    S369_M_동작_선택_8 AT %MW5040.7 : BOOL; (* S369_M_동작_선택_8 *)
    S369_M_동작_선택_9 AT %MW5040.8 : BOOL; (* S369_M_동작_선택_9 *)
    S369_M_로딩_공정_불간섭 AT %MW5004.2 : BOOL; (* S369_M_공정_불간섭 *)
    S369_M_로딩_공정_원위치 AT %MW5004.0 : BOOL; (* S369_M_공정_원위치 *)
    S369_M_로딩_리셋보조 AT %MW5000.13 : BOOL;
    S369_M_로딩_이젝터_제품감지_무 AT %MW5001.9 : BOOL;
    S369_M_로딩_이젝터_제품감지_유 AT %MW5001.8 : BOOL;
    S369_M_로딩_작업_완료 AT %MW5001.0 : BOOL; (* S369_M_작업_완료 *)
    S369_M_로딩버퍼_SEQ AT %MW10240 : WORD; (* S369 M 로딩버퍼 SEQ *)
    S369_M_로딩버퍼_VIN_NO_1_2 AT %MW10251 : WORD; (* S369 M 로딩버퍼 VIN NO 1 2 *)
    S369_M_로딩버퍼_VIN_NO_3_4 AT %MW10252 : WORD; (* S369 M 로딩버퍼 VIN NO 3 4 *)
    S369_M_로딩버퍼_VIN_NO_5_6 AT %MW10253 : WORD; (* S369 M 로딩버퍼 VIN NO 5 6 *)
    S369_M_로딩버퍼_VIN_NO_7_8 AT %MW10254 : WORD; (* S369 M 로딩버퍼 VIN NO 7 8 *)
    S369_M_로딩버퍼_VIN_NO_9_10 AT %MW10255 : WORD; (* S369 M 로딩버퍼 VIN NO 9 10 *)
    S369_M_로딩버퍼_제품감지_무 AT %MW5005.1 : BOOL; (* S369_로딩버퍼_제품감지_무 *)
    S369_M_로딩버퍼_제품감지_유 AT %MW5005.0 : BOOL; (* S369_로딩버퍼_제품감지_유 *)
    S369_M_로딩버퍼_차종1_AX AT %MW10241.0 : BOOL; (* S369 M 로딩버퍼 차종1 AX *)
    S369_M_로딩버퍼_차종1_B AT %MW10241.1 : BOOL; (* S369 M 로딩버퍼 차종1 B *)
    S369_M_로딩버퍼_차종1_C AT %MW10241.2 : BOOL; (* S369 M 로딩버퍼 차종1 C *)
    S369_M_로딩버퍼_차종1_D AT %MW10241.3 : BOOL; (* S369 M 로딩버퍼 차종1 D *)
    S369_M_로딩버퍼_차종1_E AT %MW10241.4 : BOOL; (* S369 M 로딩버퍼 차종1 E *)
    S369_M_로딩버퍼_차종1_F AT %MW10241.5 : BOOL; (* S369 M 로딩버퍼 차종1 F *)
    S369_M_로딩버퍼_차종1_G AT %MW10241.6 : BOOL; (* S369 M 로딩버퍼 차종1 G *)
    S369_M_로딩버퍼_차종1_H AT %MW10241.7 : BOOL; (* S369 M 로딩버퍼 차종1 H *)
    S369_M_로딩버퍼_차종2_3DR AT %MW10241.8 : BOOL; (* S369 M 로딩버퍼 차종2 3DR *)
    S369_M_로딩버퍼_차종2_4DR AT %MW10241.9 : BOOL; (* S369 M 로딩버퍼 차종2 4DR *)
    S369_M_로딩버퍼_차종2_5DR AT %MW10241.10 : BOOL; (* S369 M 로딩버퍼 차종2 5DR *)
    S369_M_로딩버퍼_차종2_SP1 AT %MW10241.12 : BOOL; (* S369 M 로딩버퍼 차종2 SP1 *)
    S369_M_로딩버퍼_차종2_SP2 AT %MW10241.13 : BOOL; (* S369 M 로딩버퍼 차종2 SP2 *)
    S369_M_로딩버퍼_차종2_WGN AT %MW10241.11 : BOOL; (* S369 M 로딩버퍼 차종2 WGN *)
    S369_M_로딩버퍼_차종3_LHD AT %MW10241.14 : BOOL; (* S369 M 로딩버퍼 차종3 LHD *)
    S369_M_로딩버퍼_차종3_RHD AT %MW10241.15 : BOOL; (* S369 M 로딩버퍼 차종3 RHD *)
    S369_M_로딩버퍼_차종4_EEC AT %MW10242.3 : BOOL; (* S369 M 로딩버퍼 차종4 EEC *)
    S369_M_로딩버퍼_차종4_SP1 AT %MW10242.8 : BOOL; (* S369 M 로딩버퍼 차종4 SP1 *)
    S369_M_로딩버퍼_차종4_SP2 AT %MW10242.9 : BOOL; (* S369 M 로딩버퍼 차종4 SP2 *)
    S369_M_로딩버퍼_차종4_SP3 AT %MW10242.11 : BOOL; (* S369 M 로딩버퍼 차종4 SP3 *)
    S369_M_로딩버퍼_차종4_SP4 AT %MW10242.12 : BOOL; (* S369 M 로딩버퍼 차종4 SP4 *)
    S369_M_로딩버퍼_차종4_SP5 AT %MW10242.13 : BOOL; (* S369 M 로딩버퍼 차종4 SP5 *)
    S369_M_로딩버퍼_차종4_SP6 AT %MW10242.14 : BOOL; (* S369 M 로딩버퍼 차종4 SP6 *)
    S369_M_로딩버퍼_차종4_SP7 AT %MW10242.15 : BOOL; (* S369 M 로딩버퍼 차종4 SP7 *)
    S369_M_로딩버퍼_차종4_내수 AT %MW10242.0 : BOOL; (* S369 M 로딩버퍼 차종4 내수 *)
    S369_M_로딩버퍼_차종4_러시아 AT %MW10242.10 : BOOL; (* S369 M 로딩버퍼 차종4 러시아 *)
    S369_M_로딩버퍼_차종4_북미 AT %MW10242.2 : BOOL; (* S369 M 로딩버퍼 차종4 북미 *)
    S369_M_로딩버퍼_차종4_브라질 AT %MW10242.7 : BOOL; (* S369 M 로딩버퍼 차종4 브라질 *)
    S369_M_로딩버퍼_차종4_수출 AT %MW10242.1 : BOOL; (* S369 M 로딩버퍼 차종4 수출 *)
    S369_M_로딩버퍼_차종4_중국 AT %MW10242.6 : BOOL; (* S369 M 로딩버퍼 차종4 중국 *)
    S369_M_로딩버퍼_차종4_중동 AT %MW10242.5 : BOOL; (* S369 M 로딩버퍼 차종4 중동 *)
    S369_M_로딩버퍼_차종4_호주 AT %MW10242.4 : BOOL; (* S369 M 로딩버퍼 차종4 호주 *)
    S369_M_로딩버퍼_차종5_AT AT %MW10243.1 : BOOL; (* S369 M 로딩버퍼 차종5 AT *)
    S369_M_로딩버퍼_차종5_MT AT %MW10243.0 : BOOL; (* S369 M 로딩버퍼 차종5 MT *)
    S369_M_로딩버퍼_차종5_SP1 AT %MW10243.2 : BOOL; (* S369 M 로딩버퍼 차종5 SP1 *)
    S369_M_로딩버퍼_차종6_DSROOF AT %MW10243.6 : BOOL; (* S369 M 로딩버퍼 차종6 DSROOF *)
    S369_M_로딩버퍼_차종6_SP1 AT %MW10243.7 : BOOL; (* S369 M 로딩버퍼 차종6 SP1 *)
    S369_M_로딩버퍼_차종6_썬루프 AT %MW10243.4 : BOOL; (* S369 M 로딩버퍼 차종6 썬루프 *)
    S369_M_로딩버퍼_차종6_일반루프 AT %MW10243.3 : BOOL; (* S369 M 로딩버퍼 차종6 일반루프 *)
    S369_M_로딩버퍼_차종6_파노라마루프 AT %MW10243.5 : BOOL; (* S369 M 로딩버퍼 차종6 파노라마루프 *)
    S369_M_로딩버퍼_차종7_DSL AT %MW10243.9 : BOOL; (* S369 M 로딩버퍼 차종7 DSL *)
    S369_M_로딩버퍼_차종7_GSL AT %MW10243.8 : BOOL; (* S369 M 로딩버퍼 차종7 GSL *)
    S369_M_로딩버퍼_차종7_SP1 AT %MW10243.10 : BOOL; (* S369 M 로딩버퍼 차종7 SP1 *)
    S369_M_로딩버퍼_차종7_SP2 AT %MW10243.11 : BOOL; (* S369 M 로딩버퍼 차종7 SP2 *)
    S369_M_로딩버퍼_차종7_SP3 AT %MW10243.12 : BOOL; (* S369 M 로딩버퍼 차종7 SP3 *)
    S369_M_로딩버퍼_차종7_SP4 AT %MW10243.13 : BOOL; (* S369 M 로딩버퍼 차종7 SP4 *)
    S369_M_로딩버퍼_차종7_SP5 AT %MW10243.14 : BOOL; (* S369 M 로딩버퍼 차종7 SP5 *)
    S369_M_로딩버퍼_차종7_SP6 AT %MW10243.15 : BOOL; (* S369 M 로딩버퍼 차종7 SP6 *)
    S369_M_로딩버퍼_차종8_2WD AT %MW10244.0 : BOOL; (* S369 M 로딩버퍼 차종8 2WD *)
    S369_M_로딩버퍼_차종8_4WD AT %MW10244.1 : BOOL; (* S369 M 로딩버퍼 차종8 4WD *)
    S369_M_로딩버퍼_차종8_SP1 AT %MW10244.2 : BOOL; (* S369 M 로딩버퍼 차종8 SP1 *)
    S369_M_로딩버퍼_차종9_MPI AT %MW10244.3 : BOOL; (* S369 M 로딩버퍼 차종9 MPI *)
    S369_M_로딩버퍼_차종9_SP1 AT %MW10244.5 : BOOL; (* S369 M 로딩버퍼 차종9 SP1 *)
    S369_M_로딩버퍼_차종9_SP10 AT %MW10244.14 : BOOL; (* S369 M 로딩버퍼 차종9 SP10 *)
    S369_M_로딩버퍼_차종9_SP11 AT %MW10244.15 : BOOL; (* S369 M 로딩버퍼 차종9 SP11 *)
    S369_M_로딩버퍼_차종9_SP2 AT %MW10244.6 : BOOL; (* S369 M 로딩버퍼 차종9 SP2 *)
    S369_M_로딩버퍼_차종9_SP3 AT %MW10244.7 : BOOL; (* S369 M 로딩버퍼 차종9 SP3 *)
    S369_M_로딩버퍼_차종9_SP4 AT %MW10244.8 : BOOL; (* S369 M 로딩버퍼 차종9 SP4 *)
    S369_M_로딩버퍼_차종9_SP5 AT %MW10244.9 : BOOL; (* S369 M 로딩버퍼 차종9 SP5 *)
    S369_M_로딩버퍼_차종9_SP6 AT %MW10244.10 : BOOL; (* S369 M 로딩버퍼 차종9 SP6 *)
    S369_M_로딩버퍼_차종9_SP7 AT %MW10244.11 : BOOL; (* S369 M 로딩버퍼 차종9 SP7 *)
    S369_M_로딩버퍼_차종9_SP8 AT %MW10244.12 : BOOL; (* S369 M 로딩버퍼 차종9 SP8 *)
    S369_M_로딩버퍼_차종9_SP9 AT %MW10244.13 : BOOL; (* S369 M 로딩버퍼 차종9 SP9 *)
    S369_M_로딩버퍼_차종9_T_GDI AT %MW10244.4 : BOOL; (* S369 M 로딩버퍼 차종9 T GDI *)
    S369_M_로딩버퍼_차종_AS AT %MW10250.9 : BOOL; (* S369 M 로딩버퍼 차종 AS *)
    S369_M_로딩버퍼_차종_OPT1_R_RACK_무 AT %MW10245.3 : BOOL; (* S369 M 로딩버퍼 차종 OPT1 R RACK 무 *)
    S369_M_로딩버퍼_차종_OPT1_R_RACK_유 AT %MW10245.2 : BOOL; (* S369 M 로딩버퍼 차종 OPT1 R RACK 유 *)
    S369_M_로딩버퍼_차종_OPT1_SP1 AT %MW10245.10 : BOOL; (* S369 M 로딩버퍼 차종 OPT1 SP1 *)
    S369_M_로딩버퍼_차종_OPT1_SP2 AT %MW10245.11 : BOOL; (* S369 M 로딩버퍼 차종 OPT1 SP2 *)
    S369_M_로딩버퍼_차종_OPT1_SP3 AT %MW10245.12 : BOOL; (* S369 M 로딩버퍼 차종 OPT1 SP3 *)
    S369_M_로딩버퍼_차종_OPT1_SP4 AT %MW10245.13 : BOOL; (* S369 M 로딩버퍼 차종 OPT1 SP4 *)
    S369_M_로딩버퍼_차종_OPT1_SP5 AT %MW10245.14 : BOOL; (* S369 M 로딩버퍼 차종 OPT1 SP5 *)
    S369_M_로딩버퍼_차종_OPT1_SP6 AT %MW10245.15 : BOOL; (* S369 M 로딩버퍼 차종 OPT1 SP6 *)
    S369_M_로딩버퍼_차종_OPT1_S_REP_EATER_무 AT %MW10245.7 : BOOL; (* S369 M 로딩버퍼 차종 OPT1 S REP EATER 무 *)
    S369_M_로딩버퍼_차종_OPT1_S_REP_EATER_유 AT %MW10245.6 : BOOL; (* S369 M 로딩버퍼 차종 OPT1 S REP EATER 유 *)
    S369_M_로딩버퍼_차종_OPT1_VAN_무 AT %MW10245.9 : BOOL; (* S369 M 로딩버퍼 차종 OPT1 VAN 무 *)
    S369_M_로딩버퍼_차종_OPT1_VAN_유 AT %MW10245.8 : BOOL; (* S369 M 로딩버퍼 차종 OPT1 VAN 유 *)
    S369_M_로딩버퍼_차종_OPT1_슬라이딩_무 AT %MW10245.1 : BOOL; (* S369 M 로딩버퍼 차종 OPT1 슬라이딩 무 *)
    S369_M_로딩버퍼_차종_OPT1_슬라이딩_유 AT %MW10245.0 : BOOL; (* S369 M 로딩버퍼 차종 OPT1 슬라이딩 유 *)
    S369_M_로딩버퍼_차종_OPT1_폴딩_무 AT %MW10245.5 : BOOL; (* S369 M 로딩버퍼 차종 OPT1 폴딩 무 *)
    S369_M_로딩버퍼_차종_OPT1_폴딩_유 AT %MW10245.4 : BOOL; (* S369 M 로딩버퍼 차종 OPT1 폴딩 유 *)
    S369_M_로딩버퍼_차종_OPT2_SP_WORD1 AT %MW10246 : WORD; (* S369 M 로딩버퍼 차종 OPT2 SP WORD1 *)
    S369_M_로딩버퍼_차종_OPT3_SP_WORD2 AT %MW10247 : WORD; (* S369 M 로딩버퍼 차종 OPT3 SP WORD2 *)
    S369_M_로딩버퍼_차종_OPT4_SP_WORD3 AT %MW10248 : WORD; (* S369 M 로딩버퍼 차종 OPT4 SP WORD3 *)
    S369_M_로딩버퍼_차종_OPT5_SP_WORD4 AT %MW10249 : WORD; (* S369 M 로딩버퍼 차종 OPT5 SP WORD4 *)
    S369_M_로딩버퍼_차종_SP1 AT %MW10250.0 : BOOL; (* S369 M 로딩버퍼 차종 SP1 *)
    S369_M_로딩버퍼_차종_SP2 AT %MW10250.1 : BOOL; (* S369 M 로딩버퍼 차종 SP2 *)
    S369_M_로딩버퍼_차종_SP3 AT %MW10250.2 : BOOL; (* S369 M 로딩버퍼 차종 SP3 *)
    S369_M_로딩버퍼_차종_SP4 AT %MW10250.3 : BOOL; (* S369 M 로딩버퍼 차종 SP4 *)
    S369_M_로딩버퍼_차종_SP5 AT %MW10250.4 : BOOL; (* S369 M 로딩버퍼 차종 SP5 *)
    S369_M_로딩버퍼_차종_SP6 AT %MW10250.5 : BOOL; (* S369 M 로딩버퍼 차종 SP6 *)
    S369_M_로딩버퍼_차종_SP7 AT %MW10250.6 : BOOL; (* S369 M 로딩버퍼 차종 SP7 *)
    S369_M_로딩버퍼_차종_SP8 AT %MW10250.7 : BOOL; (* S369 M 로딩버퍼 차종 SP8 *)
    S369_M_로딩버퍼_차종_SP9 AT %MW10250.15 : BOOL; (* S369 M 로딩버퍼 차종 SP9 *)
    S369_M_로딩버퍼_차종_공대차 AT %MW10250.12 : BOOL; (* S369 M 로딩버퍼 차종 공대차 *)
    S369_M_로딩버퍼_차종_공차 AT %MW10250.10 : BOOL; (* S369 M 로딩버퍼 차종 공차 *)
    S369_M_로딩버퍼_차종_무 AT %MW5002.1 : BOOL;
    S369_M_로딩버퍼_차종_불량대차 AT %MW10250.13 : BOOL; (* S369 M 로딩버퍼 차종 불량대차 *)
    S369_M_로딩버퍼_차종_불량차 AT %MW10250.11 : BOOL; (* S369 M 로딩버퍼 차종 불량차 *)
    S369_M_로딩버퍼_차종_비축 AT %MW10250.8 : BOOL; (* S369 M 로딩버퍼 차종 비축 *)
    S369_M_로딩버퍼_차종_유 AT %MW5002.0 : BOOL;
    S369_M_로딩버퍼_차종_취출대차 AT %MW10250.14 : BOOL; (* S369 M 로딩버퍼 차종 취출대차 *)
    S369_M_부저_정지_보조 AT %MW5000.11 : BOOL; (* S369_M_부저_정지_보조 *)
    S369_M_수동모드 AT %MW5000.3 : BOOL; (* S369 선택 수동모드 *)
    S369_M_언로딩_공정_불간섭 AT %MW5004.3 : BOOL;
    S369_M_언로딩_공정_원위치 AT %MW5004.1 : BOOL;
    S369_M_언로딩_이젝터_제품감지_무 AT %MW5001.11 : BOOL;
    S369_M_언로딩_이젝터_제품감지_유 AT %MW5001.10 : BOOL;
    S369_M_언로딩_작업_완료 AT %MW5001.1 : BOOL;
    S369_M_언로딩버퍼_SEQ AT %MW10340 : WORD; (* S369 M 언로딩버퍼 SEQ *)
    S369_M_언로딩버퍼_VIN_NO_1_2 AT %MW10351 : WORD; (* S369 M 언로딩버퍼 VIN NO 1 2 *)
    S369_M_언로딩버퍼_VIN_NO_3_4 AT %MW10352 : WORD; (* S369 M 언로딩버퍼 VIN NO 3 4 *)
    S369_M_언로딩버퍼_VIN_NO_5_6 AT %MW10353 : WORD; (* S369 M 언로딩버퍼 VIN NO 5 6 *)
    S369_M_언로딩버퍼_VIN_NO_7_8 AT %MW10354 : WORD; (* S369 M 언로딩버퍼 VIN NO 7 8 *)
    S369_M_언로딩버퍼_VIN_NO_9_10 AT %MW10355 : WORD; (* S369 M 언로딩버퍼 VIN NO 9 10 *)
    S369_M_언로딩버퍼_도착완료 AT %MW5003.6 : BOOL;
    S369_M_언로딩버퍼_제품감지_무 AT %MW5005.11 : BOOL; (* S369_언로딩버퍼_제품감지_무 *)
    S369_M_언로딩버퍼_제품감지_유 AT %MW5005.10 : BOOL; (* S369_언로딩버퍼_제품감지_유 *)
    S369_M_언로딩버퍼_차종1_AX AT %MW10341.0 : BOOL; (* S369 M 언로딩버퍼 차종1 AX *)
    S369_M_언로딩버퍼_차종1_B AT %MW10341.1 : BOOL; (* S369 M 언로딩버퍼 차종1 B *)
    S369_M_언로딩버퍼_차종1_C AT %MW10341.2 : BOOL; (* S369 M 언로딩버퍼 차종1 C *)
    S369_M_언로딩버퍼_차종1_D AT %MW10341.3 : BOOL; (* S369 M 언로딩버퍼 차종1 D *)
    S369_M_언로딩버퍼_차종1_E AT %MW10341.4 : BOOL; (* S369 M 언로딩버퍼 차종1 E *)
    S369_M_언로딩버퍼_차종1_F AT %MW10341.5 : BOOL; (* S369 M 언로딩버퍼 차종1 F *)
    S369_M_언로딩버퍼_차종1_G AT %MW10341.6 : BOOL; (* S369 M 언로딩버퍼 차종1 G *)
    S369_M_언로딩버퍼_차종1_H AT %MW10341.7 : BOOL; (* S369 M 언로딩버퍼 차종1 H *)
    S369_M_언로딩버퍼_차종2_3DR AT %MW10341.8 : BOOL; (* S369 M 언로딩버퍼 차종2 3DR *)
    S369_M_언로딩버퍼_차종2_4DR AT %MW10341.9 : BOOL; (* S369 M 언로딩버퍼 차종2 4DR *)
    S369_M_언로딩버퍼_차종2_5DR AT %MW10341.10 : BOOL; (* S369 M 언로딩버퍼 차종2 5DR *)
    S369_M_언로딩버퍼_차종2_SP1 AT %MW10341.12 : BOOL; (* S369 M 언로딩버퍼 차종2 SP1 *)
    S369_M_언로딩버퍼_차종2_SP2 AT %MW10341.13 : BOOL; (* S369 M 언로딩버퍼 차종2 SP2 *)
    S369_M_언로딩버퍼_차종2_WGN AT %MW10341.11 : BOOL; (* S369 M 언로딩버퍼 차종2 WGN *)
    S369_M_언로딩버퍼_차종3_LHD AT %MW10341.14 : BOOL; (* S369 M 언로딩버퍼 차종3 LHD *)
    S369_M_언로딩버퍼_차종3_RHD AT %MW10341.15 : BOOL; (* S369 M 언로딩버퍼 차종3 RHD *)
    S369_M_언로딩버퍼_차종4_EEC AT %MW10342.3 : BOOL; (* S369 M 언로딩버퍼 차종4 EEC *)
    S369_M_언로딩버퍼_차종4_SP1 AT %MW10342.8 : BOOL; (* S369 M 언로딩버퍼 차종4 SP1 *)
    S369_M_언로딩버퍼_차종4_SP2 AT %MW10342.9 : BOOL; (* S369 M 언로딩버퍼 차종4 SP2 *)
    S369_M_언로딩버퍼_차종4_SP3 AT %MW10342.11 : BOOL; (* S369 M 언로딩버퍼 차종4 SP3 *)
    S369_M_언로딩버퍼_차종4_SP4 AT %MW10342.12 : BOOL; (* S369 M 언로딩버퍼 차종4 SP4 *)
    S369_M_언로딩버퍼_차종4_SP5 AT %MW10342.13 : BOOL; (* S369 M 언로딩버퍼 차종4 SP5 *)
    S369_M_언로딩버퍼_차종4_SP6 AT %MW10342.14 : BOOL; (* S369 M 언로딩버퍼 차종4 SP6 *)
    S369_M_언로딩버퍼_차종4_SP7 AT %MW10342.15 : BOOL; (* S369 M 언로딩버퍼 차종4 SP7 *)
    S369_M_언로딩버퍼_차종4_내수 AT %MW10342.0 : BOOL; (* S369 M 언로딩버퍼 차종4 내수 *)
    S369_M_언로딩버퍼_차종4_러시아 AT %MW10342.10 : BOOL; (* S369 M 언로딩버퍼 차종4 러시아 *)
    S369_M_언로딩버퍼_차종4_북미 AT %MW10342.2 : BOOL; (* S369 M 언로딩버퍼 차종4 북미 *)
    S369_M_언로딩버퍼_차종4_브라질 AT %MW10342.7 : BOOL; (* S369 M 언로딩버퍼 차종4 브라질 *)
    S369_M_언로딩버퍼_차종4_수출 AT %MW10342.1 : BOOL; (* S369 M 언로딩버퍼 차종4 수출 *)
    S369_M_언로딩버퍼_차종4_중국 AT %MW10342.6 : BOOL; (* S369 M 언로딩버퍼 차종4 중국 *)
    S369_M_언로딩버퍼_차종4_중동 AT %MW10342.5 : BOOL; (* S369 M 언로딩버퍼 차종4 중동 *)
    S369_M_언로딩버퍼_차종4_호주 AT %MW10342.4 : BOOL; (* S369 M 언로딩버퍼 차종4 호주 *)
    S369_M_언로딩버퍼_차종5_AT AT %MW10343.1 : BOOL; (* S369 M 언로딩버퍼 차종5 AT *)
    S369_M_언로딩버퍼_차종5_MT AT %MW10343.0 : BOOL; (* S369 M 언로딩버퍼 차종5 MT *)
    S369_M_언로딩버퍼_차종5_SP1 AT %MW10343.2 : BOOL; (* S369 M 언로딩버퍼 차종5 SP1 *)
    S369_M_언로딩버퍼_차종6_DSROOF AT %MW10343.6 : BOOL; (* S369 M 언로딩버퍼 차종6 DSROOF *)
    S369_M_언로딩버퍼_차종6_SP1 AT %MW10343.7 : BOOL; (* S369 M 언로딩버퍼 차종6 SP1 *)
    S369_M_언로딩버퍼_차종6_썬루프 AT %MW10343.4 : BOOL; (* S369 M 언로딩버퍼 차종6 썬루프 *)
    S369_M_언로딩버퍼_차종6_일반루프 AT %MW10343.3 : BOOL; (* S369 M 언로딩버퍼 차종6 일반루프 *)
    S369_M_언로딩버퍼_차종6_파노라마루프 AT %MW10343.5 : BOOL; (* S369 M 언로딩버퍼 차종6 파노라마루프 *)
    S369_M_언로딩버퍼_차종7_DSL AT %MW10343.9 : BOOL; (* S369 M 언로딩버퍼 차종7 DSL *)
    S369_M_언로딩버퍼_차종7_GSL AT %MW10343.8 : BOOL; (* S369 M 언로딩버퍼 차종7 GSL *)
    S369_M_언로딩버퍼_차종7_SP1 AT %MW10343.10 : BOOL; (* S369 M 언로딩버퍼 차종7 SP1 *)
    S369_M_언로딩버퍼_차종7_SP2 AT %MW10343.11 : BOOL; (* S369 M 언로딩버퍼 차종7 SP2 *)
    S369_M_언로딩버퍼_차종7_SP3 AT %MW10343.12 : BOOL; (* S369 M 언로딩버퍼 차종7 SP3 *)
    S369_M_언로딩버퍼_차종7_SP4 AT %MW10343.13 : BOOL; (* S369 M 언로딩버퍼 차종7 SP4 *)
    S369_M_언로딩버퍼_차종7_SP5 AT %MW10343.14 : BOOL; (* S369 M 언로딩버퍼 차종7 SP5 *)
    S369_M_언로딩버퍼_차종7_SP6 AT %MW10343.15 : BOOL; (* S369 M 언로딩버퍼 차종7 SP6 *)
    S369_M_언로딩버퍼_차종8_2WD AT %MW10344.0 : BOOL; (* S369 M 언로딩버퍼 차종8 2WD *)
    S369_M_언로딩버퍼_차종8_4WD AT %MW10344.1 : BOOL; (* S369 M 언로딩버퍼 차종8 4WD *)
    S369_M_언로딩버퍼_차종8_SP1 AT %MW10344.2 : BOOL; (* S369 M 언로딩버퍼 차종8 SP1 *)
    S369_M_언로딩버퍼_차종9_MPI AT %MW10344.3 : BOOL; (* S369 M 언로딩버퍼 차종9 MPI *)
    S369_M_언로딩버퍼_차종9_SP1 AT %MW10344.5 : BOOL; (* S369 M 언로딩버퍼 차종9 SP1 *)
    S369_M_언로딩버퍼_차종9_SP10 AT %MW10344.14 : BOOL; (* S369 M 언로딩버퍼 차종9 SP10 *)
    S369_M_언로딩버퍼_차종9_SP11 AT %MW10344.15 : BOOL; (* S369 M 언로딩버퍼 차종9 SP11 *)
    S369_M_언로딩버퍼_차종9_SP2 AT %MW10344.6 : BOOL; (* S369 M 언로딩버퍼 차종9 SP2 *)
    S369_M_언로딩버퍼_차종9_SP3 AT %MW10344.7 : BOOL; (* S369 M 언로딩버퍼 차종9 SP3 *)
    S369_M_언로딩버퍼_차종9_SP4 AT %MW10344.8 : BOOL; (* S369 M 언로딩버퍼 차종9 SP4 *)
    S369_M_언로딩버퍼_차종9_SP5 AT %MW10344.9 : BOOL; (* S369 M 언로딩버퍼 차종9 SP5 *)
    S369_M_언로딩버퍼_차종9_SP6 AT %MW10344.10 : BOOL; (* S369 M 언로딩버퍼 차종9 SP6 *)
    S369_M_언로딩버퍼_차종9_SP7 AT %MW10344.11 : BOOL; (* S369 M 언로딩버퍼 차종9 SP7 *)
    S369_M_언로딩버퍼_차종9_SP8 AT %MW10344.12 : BOOL; (* S369 M 언로딩버퍼 차종9 SP8 *)
    S369_M_언로딩버퍼_차종9_SP9 AT %MW10344.13 : BOOL; (* S369 M 언로딩버퍼 차종9 SP9 *)
    S369_M_언로딩버퍼_차종9_T_GDI AT %MW10344.4 : BOOL; (* S369 M 언로딩버퍼 차종9 T GDI *)
    S369_M_언로딩버퍼_차종_AS AT %MW10350.9 : BOOL; (* S369 M 언로딩버퍼 차종 AS *)
    S369_M_언로딩버퍼_차종_OPT1_R_RACK_무 AT %MW10345.3 : BOOL; (* S369 M 언로딩버퍼 차종 OPT1 R RACK 무 *)
    S369_M_언로딩버퍼_차종_OPT1_R_RACK_유 AT %MW10345.2 : BOOL; (* S369 M 언로딩버퍼 차종 OPT1 R RACK 유 *)
    S369_M_언로딩버퍼_차종_OPT1_SP1 AT %MW10345.10 : BOOL; (* S369 M 언로딩버퍼 차종 OPT1 SP1 *)
    S369_M_언로딩버퍼_차종_OPT1_SP2 AT %MW10345.11 : BOOL; (* S369 M 언로딩버퍼 차종 OPT1 SP2 *)
    S369_M_언로딩버퍼_차종_OPT1_SP3 AT %MW10345.12 : BOOL; (* S369 M 언로딩버퍼 차종 OPT1 SP3 *)
    S369_M_언로딩버퍼_차종_OPT1_SP4 AT %MW10345.13 : BOOL; (* S369 M 언로딩버퍼 차종 OPT1 SP4 *)
    S369_M_언로딩버퍼_차종_OPT1_SP5 AT %MW10345.14 : BOOL; (* S369 M 언로딩버퍼 차종 OPT1 SP5 *)
    S369_M_언로딩버퍼_차종_OPT1_SP6 AT %MW10345.15 : BOOL; (* S369 M 언로딩버퍼 차종 OPT1 SP6 *)
    S369_M_언로딩버퍼_차종_OPT1_S_REP_EATER_무 AT %MW10345.7 : BOOL; (* S369 M 언로딩버퍼 차종 OPT1 S REP EATER 무 *)
    S369_M_언로딩버퍼_차종_OPT1_S_REP_EATER_유 AT %MW10345.6 : BOOL; (* S369 M 언로딩버퍼 차종 OPT1 S REP EATER 유 *)
    S369_M_언로딩버퍼_차종_OPT1_VAN_무 AT %MW10345.9 : BOOL; (* S369 M 언로딩버퍼 차종 OPT1 VAN 무 *)
    S369_M_언로딩버퍼_차종_OPT1_VAN_유 AT %MW10345.8 : BOOL; (* S369 M 언로딩버퍼 차종 OPT1 VAN 유 *)
    S369_M_언로딩버퍼_차종_OPT1_슬라이딩_무 AT %MW10345.1 : BOOL; (* S369 M 언로딩버퍼 차종 OPT1 슬라이딩 무 *)
    S369_M_언로딩버퍼_차종_OPT1_슬라이딩_유 AT %MW10345.0 : BOOL; (* S369 M 언로딩버퍼 차종 OPT1 슬라이딩 유 *)
    S369_M_언로딩버퍼_차종_OPT1_폴딩_무 AT %MW10345.5 : BOOL; (* S369 M 언로딩버퍼 차종 OPT1 폴딩 무 *)
    S369_M_언로딩버퍼_차종_OPT1_폴딩_유 AT %MW10345.4 : BOOL; (* S369 M 언로딩버퍼 차종 OPT1 폴딩 유 *)
    S369_M_언로딩버퍼_차종_OPT2_SP_WORD1 AT %MW10346 : WORD; (* S369 M 언로딩버퍼 차종 OPT2 SP WORD1 *)
    S369_M_언로딩버퍼_차종_OPT3_SP_WORD2 AT %MW10347 : WORD; (* S369 M 언로딩버퍼 차종 OPT3 SP WORD2 *)
    S369_M_언로딩버퍼_차종_OPT4_SP_WORD3 AT %MW10348 : WORD; (* S369 M 언로딩버퍼 차종 OPT4 SP WORD3 *)
    S369_M_언로딩버퍼_차종_OPT5_SP_WORD4 AT %MW10349 : WORD; (* S369 M 언로딩버퍼 차종 OPT5 SP WORD4 *)
    S369_M_언로딩버퍼_차종_SP1 AT %MW10350.0 : BOOL; (* S369 M 언로딩버퍼 차종 SP1 *)
    S369_M_언로딩버퍼_차종_SP2 AT %MW10350.1 : BOOL; (* S369 M 언로딩버퍼 차종 SP2 *)
    S369_M_언로딩버퍼_차종_SP3 AT %MW10350.2 : BOOL; (* S369 M 언로딩버퍼 차종 SP3 *)
    S369_M_언로딩버퍼_차종_SP4 AT %MW10350.3 : BOOL; (* S369 M 언로딩버퍼 차종 SP4 *)
    S369_M_언로딩버퍼_차종_SP5 AT %MW10350.4 : BOOL; (* S369 M 언로딩버퍼 차종 SP5 *)
    S369_M_언로딩버퍼_차종_SP6 AT %MW10350.5 : BOOL; (* S369 M 언로딩버퍼 차종 SP6 *)
    S369_M_언로딩버퍼_차종_SP7 AT %MW10350.6 : BOOL; (* S369 M 언로딩버퍼 차종 SP7 *)
    S369_M_언로딩버퍼_차종_SP8 AT %MW10350.7 : BOOL; (* S369 M 언로딩버퍼 차종 SP8 *)
    S369_M_언로딩버퍼_차종_SP9 AT %MW10350.15 : BOOL; (* S369 M 언로딩버퍼 차종 SP9 *)
    S369_M_언로딩버퍼_차종_공대차 AT %MW10350.12 : BOOL; (* S369 M 언로딩버퍼 차종 공대차 *)
    S369_M_언로딩버퍼_차종_공차 AT %MW10350.10 : BOOL; (* S369 M 언로딩버퍼 차종 공차 *)
    S369_M_언로딩버퍼_차종_무 AT %MW5002.3 : BOOL;
    S369_M_언로딩버퍼_차종_불량대차 AT %MW10350.13 : BOOL; (* S369 M 언로딩버퍼 차종 불량대차 *)
    S369_M_언로딩버퍼_차종_불량차 AT %MW10350.11 : BOOL; (* S369 M 언로딩버퍼 차종 불량차 *)
    S369_M_언로딩버퍼_차종_비축 AT %MW10350.8 : BOOL; (* S369 M 언로딩버퍼 차종 비축 *)
    S369_M_언로딩버퍼_차종_유 AT %MW5002.2 : BOOL;
    S369_M_언로딩버퍼_차종_취출대차 AT %MW10350.14 : BOOL; (* S369 M 언로딩버퍼 차종 취출대차 *)
    S369_M_운전준비_ON AT %MW5000.0 : BOOL; (* S369 운전준비 ON *)
    S369_M_이상_리셋_보조 AT %MW5000.10 : BOOL; (* S369_M_이상_리셋_보조 *)
    S369_M_이송버퍼01_제품감지_무 AT %MW5005.9 : BOOL; (* S369_이송버퍼01_제품감지_OFF *)
    S369_M_이송버퍼01_제품감지_유 AT %MW5005.8 : BOOL; (* S369_이송버퍼01_제품감지_ON *)
    S369_M_이송버퍼02_제품감지_무 AT %MW5005.7 : BOOL; (* S369_이송버퍼02_제품감지_OFF *)
    S369_M_이송버퍼02_제품감지_유 AT %MW5005.6 : BOOL; (* S369_이송버퍼02_제품감지_ON *)
    S369_M_이송버퍼03_제품감지_무 AT %MW5005.5 : BOOL; (* S369_이송버퍼03_제품감지_OFF *)
    S369_M_이송버퍼03_제품감지_유 AT %MW5005.4 : BOOL; (* S369_이송버퍼03_제품감지_ON *)
    S369_M_이송버퍼04_제품감지_무 AT %MW5005.3 : BOOL; (* S369_이송버퍼04_제품감지_OFF *)
    S369_M_이송버퍼04_제품감지_유 AT %MW5005.2 : BOOL; (* S369_이송버퍼04_제품감지_ON *)
    S369_M_이송버퍼1_SEQ AT %MW10320 : WORD; (* S369 M 이송버퍼1 SEQ *)
    S369_M_이송버퍼1_VIN_NO_1_2 AT %MW10331 : WORD; (* S369 M 이송버퍼1 VIN NO 1 2 *)
    S369_M_이송버퍼1_VIN_NO_3_4 AT %MW10332 : WORD; (* S369 M 이송버퍼1 VIN NO 3 4 *)
    S369_M_이송버퍼1_VIN_NO_5_6 AT %MW10333 : WORD; (* S369 M 이송버퍼1 VIN NO 5 6 *)
    S369_M_이송버퍼1_VIN_NO_7_8 AT %MW10334 : WORD; (* S369 M 이송버퍼1 VIN NO 7 8 *)
    S369_M_이송버퍼1_VIN_NO_9_10 AT %MW10335 : WORD; (* S369 M 이송버퍼1 VIN NO 9 10 *)
    S369_M_이송버퍼1_도착완료 AT %MW5003.5 : BOOL;
    S369_M_이송버퍼1_제품감지_이상 AT %MW5014.5 : BOOL; (* S369_M_BELT4_제품감지_이상 *)
    S369_M_이송버퍼1_차종1_AX AT %MW10321.0 : BOOL; (* S369 M 이송버퍼1 차종1 AX *)
    S369_M_이송버퍼1_차종1_B AT %MW10321.1 : BOOL; (* S369 M 이송버퍼1 차종1 B *)
    S369_M_이송버퍼1_차종1_C AT %MW10321.2 : BOOL; (* S369 M 이송버퍼1 차종1 C *)
    S369_M_이송버퍼1_차종1_D AT %MW10321.3 : BOOL; (* S369 M 이송버퍼1 차종1 D *)
    S369_M_이송버퍼1_차종1_E AT %MW10321.4 : BOOL; (* S369 M 이송버퍼1 차종1 E *)
    S369_M_이송버퍼1_차종1_F AT %MW10321.5 : BOOL; (* S369 M 이송버퍼1 차종1 F *)
    S369_M_이송버퍼1_차종1_G AT %MW10321.6 : BOOL; (* S369 M 이송버퍼1 차종1 G *)
    S369_M_이송버퍼1_차종1_H AT %MW10321.7 : BOOL; (* S369 M 이송버퍼1 차종1 H *)
    S369_M_이송버퍼1_차종2_3DR AT %MW10321.8 : BOOL; (* S369 M 이송버퍼1 차종2 3DR *)
    S369_M_이송버퍼1_차종2_4DR AT %MW10321.9 : BOOL; (* S369 M 이송버퍼1 차종2 4DR *)
    S369_M_이송버퍼1_차종2_5DR AT %MW10321.10 : BOOL; (* S369 M 이송버퍼1 차종2 5DR *)
    S369_M_이송버퍼1_차종2_SP1 AT %MW10321.12 : BOOL; (* S369 M 이송버퍼1 차종2 SP1 *)
    S369_M_이송버퍼1_차종2_SP2 AT %MW10321.13 : BOOL; (* S369 M 이송버퍼1 차종2 SP2 *)
    S369_M_이송버퍼1_차종2_WGN AT %MW10321.11 : BOOL; (* S369 M 이송버퍼1 차종2 WGN *)
    S369_M_이송버퍼1_차종3_LHD AT %MW10321.14 : BOOL; (* S369 M 이송버퍼1 차종3 LHD *)
    S369_M_이송버퍼1_차종3_RHD AT %MW10321.15 : BOOL; (* S369 M 이송버퍼1 차종3 RHD *)
    S369_M_이송버퍼1_차종4_EEC AT %MW10322.3 : BOOL; (* S369 M 이송버퍼1 차종4 EEC *)
    S369_M_이송버퍼1_차종4_SP1 AT %MW10322.8 : BOOL; (* S369 M 이송버퍼1 차종4 SP1 *)
    S369_M_이송버퍼1_차종4_SP2 AT %MW10322.9 : BOOL; (* S369 M 이송버퍼1 차종4 SP2 *)
    S369_M_이송버퍼1_차종4_SP3 AT %MW10322.11 : BOOL; (* S369 M 이송버퍼1 차종4 SP3 *)
    S369_M_이송버퍼1_차종4_SP4 AT %MW10322.12 : BOOL; (* S369 M 이송버퍼1 차종4 SP4 *)
    S369_M_이송버퍼1_차종4_SP5 AT %MW10322.13 : BOOL; (* S369 M 이송버퍼1 차종4 SP5 *)
    S369_M_이송버퍼1_차종4_SP6 AT %MW10322.14 : BOOL; (* S369 M 이송버퍼1 차종4 SP6 *)
    S369_M_이송버퍼1_차종4_SP7 AT %MW10322.15 : BOOL; (* S369 M 이송버퍼1 차종4 SP7 *)
    S369_M_이송버퍼1_차종4_내수 AT %MW10322.0 : BOOL; (* S369 M 이송버퍼1 차종4 내수 *)
    S369_M_이송버퍼1_차종4_러시아 AT %MW10322.10 : BOOL; (* S369 M 이송버퍼1 차종4 러시아 *)
    S369_M_이송버퍼1_차종4_북미 AT %MW10322.2 : BOOL; (* S369 M 이송버퍼1 차종4 북미 *)
    S369_M_이송버퍼1_차종4_브라질 AT %MW10322.7 : BOOL; (* S369 M 이송버퍼1 차종4 브라질 *)
    S369_M_이송버퍼1_차종4_수출 AT %MW10322.1 : BOOL; (* S369 M 이송버퍼1 차종4 수출 *)
    S369_M_이송버퍼1_차종4_중국 AT %MW10322.6 : BOOL; (* S369 M 이송버퍼1 차종4 중국 *)
    S369_M_이송버퍼1_차종4_중동 AT %MW10322.5 : BOOL; (* S369 M 이송버퍼1 차종4 중동 *)
    S369_M_이송버퍼1_차종4_호주 AT %MW10322.4 : BOOL; (* S369 M 이송버퍼1 차종4 호주 *)
    S369_M_이송버퍼1_차종5_AT AT %MW10323.1 : BOOL; (* S369 M 이송버퍼1 차종5 AT *)
    S369_M_이송버퍼1_차종5_MT AT %MW10323.0 : BOOL; (* S369 M 이송버퍼1 차종5 MT *)
    S369_M_이송버퍼1_차종5_SP1 AT %MW10323.2 : BOOL; (* S369 M 이송버퍼1 차종5 SP1 *)
    S369_M_이송버퍼1_차종6_DSROOF AT %MW10323.6 : BOOL; (* S369 M 이송버퍼1 차종6 DSROOF *)
    S369_M_이송버퍼1_차종6_SP1 AT %MW10323.7 : BOOL; (* S369 M 이송버퍼1 차종6 SP1 *)
    S369_M_이송버퍼1_차종6_썬루프 AT %MW10323.4 : BOOL; (* S369 M 이송버퍼1 차종6 썬루프 *)
    S369_M_이송버퍼1_차종6_일반루프 AT %MW10323.3 : BOOL; (* S369 M 이송버퍼1 차종6 일반루프 *)
    S369_M_이송버퍼1_차종6_파노라마루프 AT %MW10323.5 : BOOL; (* S369 M 이송버퍼1 차종6 파노라마루프 *)
    S369_M_이송버퍼1_차종7_DSL AT %MW10323.9 : BOOL; (* S369 M 이송버퍼1 차종7 DSL *)
    S369_M_이송버퍼1_차종7_GSL AT %MW10323.8 : BOOL; (* S369 M 이송버퍼1 차종7 GSL *)
    S369_M_이송버퍼1_차종7_SP1 AT %MW10323.10 : BOOL; (* S369 M 이송버퍼1 차종7 SP1 *)
    S369_M_이송버퍼1_차종7_SP2 AT %MW10323.11 : BOOL; (* S369 M 이송버퍼1 차종7 SP2 *)
    S369_M_이송버퍼1_차종7_SP3 AT %MW10323.12 : BOOL; (* S369 M 이송버퍼1 차종7 SP3 *)
    S369_M_이송버퍼1_차종7_SP4 AT %MW10323.13 : BOOL; (* S369 M 이송버퍼1 차종7 SP4 *)
    S369_M_이송버퍼1_차종7_SP5 AT %MW10323.14 : BOOL; (* S369 M 이송버퍼1 차종7 SP5 *)
    S369_M_이송버퍼1_차종7_SP6 AT %MW10323.15 : BOOL; (* S369 M 이송버퍼1 차종7 SP6 *)
    S369_M_이송버퍼1_차종8_2WD AT %MW10324.0 : BOOL; (* S369 M 이송버퍼1 차종8 2WD *)
    S369_M_이송버퍼1_차종8_4WD AT %MW10324.1 : BOOL; (* S369 M 이송버퍼1 차종8 4WD *)
    S369_M_이송버퍼1_차종8_SP1 AT %MW10324.2 : BOOL; (* S369 M 이송버퍼1 차종8 SP1 *)
    S369_M_이송버퍼1_차종9_MPI AT %MW10324.3 : BOOL; (* S369 M 이송버퍼1 차종9 MPI *)
    S369_M_이송버퍼1_차종9_SP1 AT %MW10324.5 : BOOL; (* S369 M 이송버퍼1 차종9 SP1 *)
    S369_M_이송버퍼1_차종9_SP10 AT %MW10324.14 : BOOL; (* S369 M 이송버퍼1 차종9 SP10 *)
    S369_M_이송버퍼1_차종9_SP11 AT %MW10324.15 : BOOL; (* S369 M 이송버퍼1 차종9 SP11 *)
    S369_M_이송버퍼1_차종9_SP2 AT %MW10324.6 : BOOL; (* S369 M 이송버퍼1 차종9 SP2 *)
    S369_M_이송버퍼1_차종9_SP3 AT %MW10324.7 : BOOL; (* S369 M 이송버퍼1 차종9 SP3 *)
    S369_M_이송버퍼1_차종9_SP4 AT %MW10324.8 : BOOL; (* S369 M 이송버퍼1 차종9 SP4 *)
    S369_M_이송버퍼1_차종9_SP5 AT %MW10324.9 : BOOL; (* S369 M 이송버퍼1 차종9 SP5 *)
    S369_M_이송버퍼1_차종9_SP6 AT %MW10324.10 : BOOL; (* S369 M 이송버퍼1 차종9 SP6 *)
    S369_M_이송버퍼1_차종9_SP7 AT %MW10324.11 : BOOL; (* S369 M 이송버퍼1 차종9 SP7 *)
    S369_M_이송버퍼1_차종9_SP8 AT %MW10324.12 : BOOL; (* S369 M 이송버퍼1 차종9 SP8 *)
    S369_M_이송버퍼1_차종9_SP9 AT %MW10324.13 : BOOL; (* S369 M 이송버퍼1 차종9 SP9 *)
    S369_M_이송버퍼1_차종9_T_GDI AT %MW10324.4 : BOOL; (* S369 M 이송버퍼1 차종9 T GDI *)
    S369_M_이송버퍼1_차종_AS AT %MW10330.9 : BOOL; (* S369 M 이송버퍼1 차종 AS *)
    S369_M_이송버퍼1_차종_OPT1_R_RACK_무 AT %MW10325.3 : BOOL; (* S369 M 이송버퍼1 차종 OPT1 R RACK 무 *)
    S369_M_이송버퍼1_차종_OPT1_R_RACK_유 AT %MW10325.2 : BOOL; (* S369 M 이송버퍼1 차종 OPT1 R RACK 유 *)
    S369_M_이송버퍼1_차종_OPT1_SP1 AT %MW10325.10 : BOOL; (* S369 M 이송버퍼1 차종 OPT1 SP1 *)
    S369_M_이송버퍼1_차종_OPT1_SP2 AT %MW10325.11 : BOOL; (* S369 M 이송버퍼1 차종 OPT1 SP2 *)
    S369_M_이송버퍼1_차종_OPT1_SP3 AT %MW10325.12 : BOOL; (* S369 M 이송버퍼1 차종 OPT1 SP3 *)
    S369_M_이송버퍼1_차종_OPT1_SP4 AT %MW10325.13 : BOOL; (* S369 M 이송버퍼1 차종 OPT1 SP4 *)
    S369_M_이송버퍼1_차종_OPT1_SP5 AT %MW10325.14 : BOOL; (* S369 M 이송버퍼1 차종 OPT1 SP5 *)
    S369_M_이송버퍼1_차종_OPT1_SP6 AT %MW10325.15 : BOOL; (* S369 M 이송버퍼1 차종 OPT1 SP6 *)
    S369_M_이송버퍼1_차종_OPT1_S_REP_EATER_무 AT %MW10325.7 : BOOL; (* S369 M 이송버퍼1 차종 OPT1 S REP EATER 무 *)
    S369_M_이송버퍼1_차종_OPT1_S_REP_EATER_유 AT %MW10325.6 : BOOL; (* S369 M 이송버퍼1 차종 OPT1 S REP EATER 유 *)
    S369_M_이송버퍼1_차종_OPT1_VAN_무 AT %MW10325.9 : BOOL; (* S369 M 이송버퍼1 차종 OPT1 VAN 무 *)
    S369_M_이송버퍼1_차종_OPT1_VAN_유 AT %MW10325.8 : BOOL; (* S369 M 이송버퍼1 차종 OPT1 VAN 유 *)
    S369_M_이송버퍼1_차종_OPT1_슬라이딩_무 AT %MW10325.1 : BOOL; (* S369 M 이송버퍼1 차종 OPT1 슬라이딩 무 *)
    S369_M_이송버퍼1_차종_OPT1_슬라이딩_유 AT %MW10325.0 : BOOL; (* S369 M 이송버퍼1 차종 OPT1 슬라이딩 유 *)
    S369_M_이송버퍼1_차종_OPT1_폴딩_무 AT %MW10325.5 : BOOL; (* S369 M 이송버퍼1 차종 OPT1 폴딩 무 *)
    S369_M_이송버퍼1_차종_OPT1_폴딩_유 AT %MW10325.4 : BOOL; (* S369 M 이송버퍼1 차종 OPT1 폴딩 유 *)
    S369_M_이송버퍼1_차종_OPT2_SP_WORD1 AT %MW10326 : WORD; (* S369 M 이송버퍼1 차종 OPT2 SP WORD1 *)
    S369_M_이송버퍼1_차종_OPT3_SP_WORD2 AT %MW10327 : WORD; (* S369 M 이송버퍼1 차종 OPT3 SP WORD2 *)
    S369_M_이송버퍼1_차종_OPT4_SP_WORD3 AT %MW10328 : WORD; (* S369 M 이송버퍼1 차종 OPT4 SP WORD3 *)
    S369_M_이송버퍼1_차종_OPT5_SP_WORD4 AT %MW10329 : WORD; (* S369 M 이송버퍼1 차종 OPT5 SP WORD4 *)
    S369_M_이송버퍼1_차종_SP1 AT %MW10330.0 : BOOL; (* S369 M 이송버퍼1 차종 SP1 *)
    S369_M_이송버퍼1_차종_SP2 AT %MW10330.1 : BOOL; (* S369 M 이송버퍼1 차종 SP2 *)
    S369_M_이송버퍼1_차종_SP3 AT %MW10330.2 : BOOL; (* S369 M 이송버퍼1 차종 SP3 *)
    S369_M_이송버퍼1_차종_SP4 AT %MW10330.3 : BOOL; (* S369 M 이송버퍼1 차종 SP4 *)
    S369_M_이송버퍼1_차종_SP5 AT %MW10330.4 : BOOL; (* S369 M 이송버퍼1 차종 SP5 *)
    S369_M_이송버퍼1_차종_SP6 AT %MW10330.5 : BOOL; (* S369 M 이송버퍼1 차종 SP6 *)
    S369_M_이송버퍼1_차종_SP7 AT %MW10330.6 : BOOL; (* S369 M 이송버퍼1 차종 SP7 *)
    S369_M_이송버퍼1_차종_SP8 AT %MW10330.7 : BOOL; (* S369 M 이송버퍼1 차종 SP8 *)
    S369_M_이송버퍼1_차종_SP9 AT %MW10330.15 : BOOL; (* S369 M 이송버퍼1 차종 SP9 *)
    S369_M_이송버퍼1_차종_공대차 AT %MW10330.12 : BOOL; (* S369 M 이송버퍼1 차종 공대차 *)
    S369_M_이송버퍼1_차종_공차 AT %MW10330.10 : BOOL; (* S369 M 이송버퍼1 차종 공차 *)
    S369_M_이송버퍼1_차종_무 AT %MW5002.11 : BOOL;
    S369_M_이송버퍼1_차종_불량대차 AT %MW10330.13 : BOOL; (* S369 M 이송버퍼1 차종 불량대차 *)
    S369_M_이송버퍼1_차종_불량차 AT %MW10330.11 : BOOL; (* S369 M 이송버퍼1 차종 불량차 *)
    S369_M_이송버퍼1_차종_비축 AT %MW10330.8 : BOOL; (* S369 M 이송버퍼1 차종 비축 *)
    S369_M_이송버퍼1_차종_유 AT %MW5002.10 : BOOL;
    S369_M_이송버퍼1_차종_취출대차 AT %MW10330.14 : BOOL; (* S369 M 이송버퍼1 차종 취출대차 *)
    S369_M_이송버퍼2_SEQ AT %MW10300 : WORD; (* S369 M 이송버퍼2 SEQ *)
    S369_M_이송버퍼2_VIN_NO_1_2 AT %MW10311 : WORD; (* S369 M 이송버퍼2 VIN NO 1 2 *)
    S369_M_이송버퍼2_VIN_NO_3_4 AT %MW10312 : WORD; (* S369 M 이송버퍼2 VIN NO 3 4 *)
    S369_M_이송버퍼2_VIN_NO_5_6 AT %MW10313 : WORD; (* S369 M 이송버퍼2 VIN NO 5 6 *)
    S369_M_이송버퍼2_VIN_NO_7_8 AT %MW10314 : WORD; (* S369 M 이송버퍼2 VIN NO 7 8 *)
    S369_M_이송버퍼2_VIN_NO_9_10 AT %MW10315 : WORD; (* S369 M 이송버퍼2 VIN NO 9 10 *)
    S369_M_이송버퍼2_도착완료 AT %MW5003.4 : BOOL;
    S369_M_이송버퍼2_제품감지_이상 AT %MW5014.4 : BOOL; (* S369_M_BELT3_제품감지_이상 *)
    S369_M_이송버퍼2_차종1_AX AT %MW10301.0 : BOOL; (* S369 M 이송버퍼2 차종1 AX *)
    S369_M_이송버퍼2_차종1_B AT %MW10301.1 : BOOL; (* S369 M 이송버퍼2 차종1 B *)
    S369_M_이송버퍼2_차종1_C AT %MW10301.2 : BOOL; (* S369 M 이송버퍼2 차종1 C *)
    S369_M_이송버퍼2_차종1_D AT %MW10301.3 : BOOL; (* S369 M 이송버퍼2 차종1 D *)
    S369_M_이송버퍼2_차종1_E AT %MW10301.4 : BOOL; (* S369 M 이송버퍼2 차종1 E *)
    S369_M_이송버퍼2_차종1_F AT %MW10301.5 : BOOL; (* S369 M 이송버퍼2 차종1 F *)
    S369_M_이송버퍼2_차종1_G AT %MW10301.6 : BOOL; (* S369 M 이송버퍼2 차종1 G *)
    S369_M_이송버퍼2_차종1_H AT %MW10301.7 : BOOL; (* S369 M 이송버퍼2 차종1 H *)
    S369_M_이송버퍼2_차종2_3DR AT %MW10301.8 : BOOL; (* S369 M 이송버퍼2 차종2 3DR *)
    S369_M_이송버퍼2_차종2_4DR AT %MW10301.9 : BOOL; (* S369 M 이송버퍼2 차종2 4DR *)
    S369_M_이송버퍼2_차종2_5DR AT %MW10301.10 : BOOL; (* S369 M 이송버퍼2 차종2 5DR *)
    S369_M_이송버퍼2_차종2_SP1 AT %MW10301.12 : BOOL; (* S369 M 이송버퍼2 차종2 SP1 *)
    S369_M_이송버퍼2_차종2_SP2 AT %MW10301.13 : BOOL; (* S369 M 이송버퍼2 차종2 SP2 *)
    S369_M_이송버퍼2_차종2_WGN AT %MW10301.11 : BOOL; (* S369 M 이송버퍼2 차종2 WGN *)
    S369_M_이송버퍼2_차종3_LHD AT %MW10301.14 : BOOL; (* S369 M 이송버퍼2 차종3 LHD *)
    S369_M_이송버퍼2_차종3_RHD AT %MW10301.15 : BOOL; (* S369 M 이송버퍼2 차종3 RHD *)
    S369_M_이송버퍼2_차종4_EEC AT %MW10302.3 : BOOL; (* S369 M 이송버퍼2 차종4 EEC *)
    S369_M_이송버퍼2_차종4_SP1 AT %MW10302.8 : BOOL; (* S369 M 이송버퍼2 차종4 SP1 *)
    S369_M_이송버퍼2_차종4_SP2 AT %MW10302.9 : BOOL; (* S369 M 이송버퍼2 차종4 SP2 *)
    S369_M_이송버퍼2_차종4_SP3 AT %MW10302.11 : BOOL; (* S369 M 이송버퍼2 차종4 SP3 *)
    S369_M_이송버퍼2_차종4_SP4 AT %MW10302.12 : BOOL; (* S369 M 이송버퍼2 차종4 SP4 *)
    S369_M_이송버퍼2_차종4_SP5 AT %MW10302.13 : BOOL; (* S369 M 이송버퍼2 차종4 SP5 *)
    S369_M_이송버퍼2_차종4_SP6 AT %MW10302.14 : BOOL; (* S369 M 이송버퍼2 차종4 SP6 *)
    S369_M_이송버퍼2_차종4_SP7 AT %MW10302.15 : BOOL; (* S369 M 이송버퍼2 차종4 SP7 *)
    S369_M_이송버퍼2_차종4_내수 AT %MW10302.0 : BOOL; (* S369 M 이송버퍼2 차종4 내수 *)
    S369_M_이송버퍼2_차종4_러시아 AT %MW10302.10 : BOOL; (* S369 M 이송버퍼2 차종4 러시아 *)
    S369_M_이송버퍼2_차종4_북미 AT %MW10302.2 : BOOL; (* S369 M 이송버퍼2 차종4 북미 *)
    S369_M_이송버퍼2_차종4_브라질 AT %MW10302.7 : BOOL; (* S369 M 이송버퍼2 차종4 브라질 *)
    S369_M_이송버퍼2_차종4_수출 AT %MW10302.1 : BOOL; (* S369 M 이송버퍼2 차종4 수출 *)
    S369_M_이송버퍼2_차종4_중국 AT %MW10302.6 : BOOL; (* S369 M 이송버퍼2 차종4 중국 *)
    S369_M_이송버퍼2_차종4_중동 AT %MW10302.5 : BOOL; (* S369 M 이송버퍼2 차종4 중동 *)
    S369_M_이송버퍼2_차종4_호주 AT %MW10302.4 : BOOL; (* S369 M 이송버퍼2 차종4 호주 *)
    S369_M_이송버퍼2_차종5_AT AT %MW10303.1 : BOOL; (* S369 M 이송버퍼2 차종5 AT *)
    S369_M_이송버퍼2_차종5_MT AT %MW10303.0 : BOOL; (* S369 M 이송버퍼2 차종5 MT *)
    S369_M_이송버퍼2_차종5_SP1 AT %MW10303.2 : BOOL; (* S369 M 이송버퍼2 차종5 SP1 *)
    S369_M_이송버퍼2_차종6_DSROOF AT %MW10303.6 : BOOL; (* S369 M 이송버퍼2 차종6 DSROOF *)
    S369_M_이송버퍼2_차종6_SP1 AT %MW10303.7 : BOOL; (* S369 M 이송버퍼2 차종6 SP1 *)
    S369_M_이송버퍼2_차종6_썬루프 AT %MW10303.4 : BOOL; (* S369 M 이송버퍼2 차종6 썬루프 *)
    S369_M_이송버퍼2_차종6_일반루프 AT %MW10303.3 : BOOL; (* S369 M 이송버퍼2 차종6 일반루프 *)
    S369_M_이송버퍼2_차종6_파노라마루프 AT %MW10303.5 : BOOL; (* S369 M 이송버퍼2 차종6 파노라마루프 *)
    S369_M_이송버퍼2_차종7_DSL AT %MW10303.9 : BOOL; (* S369 M 이송버퍼2 차종7 DSL *)
    S369_M_이송버퍼2_차종7_GSL AT %MW10303.8 : BOOL; (* S369 M 이송버퍼2 차종7 GSL *)
    S369_M_이송버퍼2_차종7_SP1 AT %MW10303.10 : BOOL; (* S369 M 이송버퍼2 차종7 SP1 *)
    S369_M_이송버퍼2_차종7_SP2 AT %MW10303.11 : BOOL; (* S369 M 이송버퍼2 차종7 SP2 *)
    S369_M_이송버퍼2_차종7_SP3 AT %MW10303.12 : BOOL; (* S369 M 이송버퍼2 차종7 SP3 *)
    S369_M_이송버퍼2_차종7_SP4 AT %MW10303.13 : BOOL; (* S369 M 이송버퍼2 차종7 SP4 *)
    S369_M_이송버퍼2_차종7_SP5 AT %MW10303.14 : BOOL; (* S369 M 이송버퍼2 차종7 SP5 *)
    S369_M_이송버퍼2_차종7_SP6 AT %MW10303.15 : BOOL; (* S369 M 이송버퍼2 차종7 SP6 *)
    S369_M_이송버퍼2_차종8_2WD AT %MW10304.0 : BOOL; (* S369 M 이송버퍼2 차종8 2WD *)
    S369_M_이송버퍼2_차종8_4WD AT %MW10304.1 : BOOL; (* S369 M 이송버퍼2 차종8 4WD *)
    S369_M_이송버퍼2_차종8_SP1 AT %MW10304.2 : BOOL; (* S369 M 이송버퍼2 차종8 SP1 *)
    S369_M_이송버퍼2_차종9_MPI AT %MW10304.3 : BOOL; (* S369 M 이송버퍼2 차종9 MPI *)
    S369_M_이송버퍼2_차종9_SP1 AT %MW10304.5 : BOOL; (* S369 M 이송버퍼2 차종9 SP1 *)
    S369_M_이송버퍼2_차종9_SP10 AT %MW10304.14 : BOOL; (* S369 M 이송버퍼2 차종9 SP10 *)
    S369_M_이송버퍼2_차종9_SP11 AT %MW10304.15 : BOOL; (* S369 M 이송버퍼2 차종9 SP11 *)
    S369_M_이송버퍼2_차종9_SP2 AT %MW10304.6 : BOOL; (* S369 M 이송버퍼2 차종9 SP2 *)
    S369_M_이송버퍼2_차종9_SP3 AT %MW10304.7 : BOOL; (* S369 M 이송버퍼2 차종9 SP3 *)
    S369_M_이송버퍼2_차종9_SP4 AT %MW10304.8 : BOOL; (* S369 M 이송버퍼2 차종9 SP4 *)
    S369_M_이송버퍼2_차종9_SP5 AT %MW10304.9 : BOOL; (* S369 M 이송버퍼2 차종9 SP5 *)
    S369_M_이송버퍼2_차종9_SP6 AT %MW10304.10 : BOOL; (* S369 M 이송버퍼2 차종9 SP6 *)
    S369_M_이송버퍼2_차종9_SP7 AT %MW10304.11 : BOOL; (* S369 M 이송버퍼2 차종9 SP7 *)
    S369_M_이송버퍼2_차종9_SP8 AT %MW10304.12 : BOOL; (* S369 M 이송버퍼2 차종9 SP8 *)
    S369_M_이송버퍼2_차종9_SP9 AT %MW10304.13 : BOOL; (* S369 M 이송버퍼2 차종9 SP9 *)
    S369_M_이송버퍼2_차종9_T_GDI AT %MW10304.4 : BOOL; (* S369 M 이송버퍼2 차종9 T GDI *)
    S369_M_이송버퍼2_차종_AS AT %MW10310.9 : BOOL; (* S369 M 이송버퍼2 차종 AS *)
    S369_M_이송버퍼2_차종_OPT1_R_RACK_무 AT %MW10305.3 : BOOL; (* S369 M 이송버퍼2 차종 OPT1 R RACK 무 *)
    S369_M_이송버퍼2_차종_OPT1_R_RACK_유 AT %MW10305.2 : BOOL; (* S369 M 이송버퍼2 차종 OPT1 R RACK 유 *)
    S369_M_이송버퍼2_차종_OPT1_SP1 AT %MW10305.10 : BOOL; (* S369 M 이송버퍼2 차종 OPT1 SP1 *)
    S369_M_이송버퍼2_차종_OPT1_SP2 AT %MW10305.11 : BOOL; (* S369 M 이송버퍼2 차종 OPT1 SP2 *)
    S369_M_이송버퍼2_차종_OPT1_SP3 AT %MW10305.12 : BOOL; (* S369 M 이송버퍼2 차종 OPT1 SP3 *)
    S369_M_이송버퍼2_차종_OPT1_SP4 AT %MW10305.13 : BOOL; (* S369 M 이송버퍼2 차종 OPT1 SP4 *)
    S369_M_이송버퍼2_차종_OPT1_SP5 AT %MW10305.14 : BOOL; (* S369 M 이송버퍼2 차종 OPT1 SP5 *)
    S369_M_이송버퍼2_차종_OPT1_SP6 AT %MW10305.15 : BOOL; (* S369 M 이송버퍼2 차종 OPT1 SP6 *)
    S369_M_이송버퍼2_차종_OPT1_S_REP_EATER_무 AT %MW10305.7 : BOOL; (* S369 M 이송버퍼2 차종 OPT1 S REP EATER 무 *)
    S369_M_이송버퍼2_차종_OPT1_S_REP_EATER_유 AT %MW10305.6 : BOOL; (* S369 M 이송버퍼2 차종 OPT1 S REP EATER 유 *)
    S369_M_이송버퍼2_차종_OPT1_VAN_무 AT %MW10305.9 : BOOL; (* S369 M 이송버퍼2 차종 OPT1 VAN 무 *)
    S369_M_이송버퍼2_차종_OPT1_VAN_유 AT %MW10305.8 : BOOL; (* S369 M 이송버퍼2 차종 OPT1 VAN 유 *)
    S369_M_이송버퍼2_차종_OPT1_슬라이딩_무 AT %MW10305.1 : BOOL; (* S369 M 이송버퍼2 차종 OPT1 슬라이딩 무 *)
    S369_M_이송버퍼2_차종_OPT1_슬라이딩_유 AT %MW10305.0 : BOOL; (* S369 M 이송버퍼2 차종 OPT1 슬라이딩 유 *)
    S369_M_이송버퍼2_차종_OPT1_폴딩_무 AT %MW10305.5 : BOOL; (* S369 M 이송버퍼2 차종 OPT1 폴딩 무 *)
    S369_M_이송버퍼2_차종_OPT1_폴딩_유 AT %MW10305.4 : BOOL; (* S369 M 이송버퍼2 차종 OPT1 폴딩 유 *)
    S369_M_이송버퍼2_차종_OPT2_SP_WORD1 AT %MW10306 : WORD; (* S369 M 이송버퍼2 차종 OPT2 SP WORD1 *)
    S369_M_이송버퍼2_차종_OPT3_SP_WORD2 AT %MW10307 : WORD; (* S369 M 이송버퍼2 차종 OPT3 SP WORD2 *)
    S369_M_이송버퍼2_차종_OPT4_SP_WORD3 AT %MW10308 : WORD; (* S369 M 이송버퍼2 차종 OPT4 SP WORD3 *)
    S369_M_이송버퍼2_차종_OPT5_SP_WORD4 AT %MW10309 : WORD; (* S369 M 이송버퍼2 차종 OPT5 SP WORD4 *)
    S369_M_이송버퍼2_차종_SP1 AT %MW10310.0 : BOOL; (* S369 M 이송버퍼2 차종 SP1 *)
    S369_M_이송버퍼2_차종_SP2 AT %MW10310.1 : BOOL; (* S369 M 이송버퍼2 차종 SP2 *)
    S369_M_이송버퍼2_차종_SP3 AT %MW10310.2 : BOOL; (* S369 M 이송버퍼2 차종 SP3 *)
    S369_M_이송버퍼2_차종_SP4 AT %MW10310.3 : BOOL; (* S369 M 이송버퍼2 차종 SP4 *)
    S369_M_이송버퍼2_차종_SP5 AT %MW10310.4 : BOOL; (* S369 M 이송버퍼2 차종 SP5 *)
    S369_M_이송버퍼2_차종_SP6 AT %MW10310.5 : BOOL; (* S369 M 이송버퍼2 차종 SP6 *)
    S369_M_이송버퍼2_차종_SP7 AT %MW10310.6 : BOOL; (* S369 M 이송버퍼2 차종 SP7 *)
    S369_M_이송버퍼2_차종_SP8 AT %MW10310.7 : BOOL; (* S369 M 이송버퍼2 차종 SP8 *)
    S369_M_이송버퍼2_차종_SP9 AT %MW10310.15 : BOOL; (* S369 M 이송버퍼2 차종 SP9 *)
    S369_M_이송버퍼2_차종_공대차 AT %MW10310.12 : BOOL; (* S369 M 이송버퍼2 차종 공대차 *)
    S369_M_이송버퍼2_차종_공차 AT %MW10310.10 : BOOL; (* S369 M 이송버퍼2 차종 공차 *)
    S369_M_이송버퍼2_차종_무 AT %MW5002.9 : BOOL;
    S369_M_이송버퍼2_차종_불량대차 AT %MW10310.13 : BOOL; (* S369 M 이송버퍼2 차종 불량대차 *)
    S369_M_이송버퍼2_차종_불량차 AT %MW10310.11 : BOOL; (* S369 M 이송버퍼2 차종 불량차 *)
    S369_M_이송버퍼2_차종_비축 AT %MW10310.8 : BOOL; (* S369 M 이송버퍼2 차종 비축 *)
    S369_M_이송버퍼2_차종_유 AT %MW5002.8 : BOOL;
    S369_M_이송버퍼2_차종_취출대차 AT %MW10310.14 : BOOL; (* S369 M 이송버퍼2 차종 취출대차 *)
    S369_M_이송버퍼3_SEQ AT %MW10280 : WORD; (* S369 M 이송버퍼3 SEQ *)
    S369_M_이송버퍼3_VIN_NO_1_2 AT %MW10291 : WORD; (* S369 M 이송버퍼3 VIN NO 1 2 *)
    S369_M_이송버퍼3_VIN_NO_3_4 AT %MW10292 : WORD; (* S369 M 이송버퍼3 VIN NO 3 4 *)
    S369_M_이송버퍼3_VIN_NO_5_6 AT %MW10293 : WORD; (* S369 M 이송버퍼3 VIN NO 5 6 *)
    S369_M_이송버퍼3_VIN_NO_7_8 AT %MW10294 : WORD; (* S369 M 이송버퍼3 VIN NO 7 8 *)
    S369_M_이송버퍼3_VIN_NO_9_10 AT %MW10295 : WORD; (* S369 M 이송버퍼3 VIN NO 9 10 *)
    S369_M_이송버퍼3_도착완료 AT %MW5003.3 : BOOL;
    S369_M_이송버퍼3_제품감지_이상 AT %MW5014.3 : BOOL; (* S369_M_BELT2_제품감지_이상 *)
    S369_M_이송버퍼3_차종1_AX AT %MW10281.0 : BOOL; (* S369 M 이송버퍼3 차종1 AX *)
    S369_M_이송버퍼3_차종1_B AT %MW10281.1 : BOOL; (* S369 M 이송버퍼3 차종1 B *)
    S369_M_이송버퍼3_차종1_C AT %MW10281.2 : BOOL; (* S369 M 이송버퍼3 차종1 C *)
    S369_M_이송버퍼3_차종1_D AT %MW10281.3 : BOOL; (* S369 M 이송버퍼3 차종1 D *)
    S369_M_이송버퍼3_차종1_E AT %MW10281.4 : BOOL; (* S369 M 이송버퍼3 차종1 E *)
    S369_M_이송버퍼3_차종1_F AT %MW10281.5 : BOOL; (* S369 M 이송버퍼3 차종1 F *)
    S369_M_이송버퍼3_차종1_G AT %MW10281.6 : BOOL; (* S369 M 이송버퍼3 차종1 G *)
    S369_M_이송버퍼3_차종1_H AT %MW10281.7 : BOOL; (* S369 M 이송버퍼3 차종1 H *)
    S369_M_이송버퍼3_차종2_3DR AT %MW10281.8 : BOOL; (* S369 M 이송버퍼3 차종2 3DR *)
    S369_M_이송버퍼3_차종2_4DR AT %MW10281.9 : BOOL; (* S369 M 이송버퍼3 차종2 4DR *)
    S369_M_이송버퍼3_차종2_5DR AT %MW10281.10 : BOOL; (* S369 M 이송버퍼3 차종2 5DR *)
    S369_M_이송버퍼3_차종2_SP1 AT %MW10281.12 : BOOL; (* S369 M 이송버퍼3 차종2 SP1 *)
    S369_M_이송버퍼3_차종2_SP2 AT %MW10281.13 : BOOL; (* S369 M 이송버퍼3 차종2 SP2 *)
    S369_M_이송버퍼3_차종2_WGN AT %MW10281.11 : BOOL; (* S369 M 이송버퍼3 차종2 WGN *)
    S369_M_이송버퍼3_차종3_LHD AT %MW10281.14 : BOOL; (* S369 M 이송버퍼3 차종3 LHD *)
    S369_M_이송버퍼3_차종3_RHD AT %MW10281.15 : BOOL; (* S369 M 이송버퍼3 차종3 RHD *)
    S369_M_이송버퍼3_차종4_EEC AT %MW10282.3 : BOOL; (* S369 M 이송버퍼3 차종4 EEC *)
    S369_M_이송버퍼3_차종4_SP1 AT %MW10282.8 : BOOL; (* S369 M 이송버퍼3 차종4 SP1 *)
    S369_M_이송버퍼3_차종4_SP2 AT %MW10282.9 : BOOL; (* S369 M 이송버퍼3 차종4 SP2 *)
    S369_M_이송버퍼3_차종4_SP3 AT %MW10282.11 : BOOL; (* S369 M 이송버퍼3 차종4 SP3 *)
    S369_M_이송버퍼3_차종4_SP4 AT %MW10282.12 : BOOL; (* S369 M 이송버퍼3 차종4 SP4 *)
    S369_M_이송버퍼3_차종4_SP5 AT %MW10282.13 : BOOL; (* S369 M 이송버퍼3 차종4 SP5 *)
    S369_M_이송버퍼3_차종4_SP6 AT %MW10282.14 : BOOL; (* S369 M 이송버퍼3 차종4 SP6 *)
    S369_M_이송버퍼3_차종4_SP7 AT %MW10282.15 : BOOL; (* S369 M 이송버퍼3 차종4 SP7 *)
    S369_M_이송버퍼3_차종4_내수 AT %MW10282.0 : BOOL; (* S369 M 이송버퍼3 차종4 내수 *)
    S369_M_이송버퍼3_차종4_러시아 AT %MW10282.10 : BOOL; (* S369 M 이송버퍼3 차종4 러시아 *)
    S369_M_이송버퍼3_차종4_북미 AT %MW10282.2 : BOOL; (* S369 M 이송버퍼3 차종4 북미 *)
    S369_M_이송버퍼3_차종4_브라질 AT %MW10282.7 : BOOL; (* S369 M 이송버퍼3 차종4 브라질 *)
    S369_M_이송버퍼3_차종4_수출 AT %MW10282.1 : BOOL; (* S369 M 이송버퍼3 차종4 수출 *)
    S369_M_이송버퍼3_차종4_중국 AT %MW10282.6 : BOOL; (* S369 M 이송버퍼3 차종4 중국 *)
    S369_M_이송버퍼3_차종4_중동 AT %MW10282.5 : BOOL; (* S369 M 이송버퍼3 차종4 중동 *)
    S369_M_이송버퍼3_차종4_호주 AT %MW10282.4 : BOOL; (* S369 M 이송버퍼3 차종4 호주 *)
    S369_M_이송버퍼3_차종5_AT AT %MW10283.1 : BOOL; (* S369 M 이송버퍼3 차종5 AT *)
    S369_M_이송버퍼3_차종5_MT AT %MW10283.0 : BOOL; (* S369 M 이송버퍼3 차종5 MT *)
    S369_M_이송버퍼3_차종5_SP1 AT %MW10283.2 : BOOL; (* S369 M 이송버퍼3 차종5 SP1 *)
    S369_M_이송버퍼3_차종6_DSROOF AT %MW10283.6 : BOOL; (* S369 M 이송버퍼3 차종6 DSROOF *)
    S369_M_이송버퍼3_차종6_SP1 AT %MW10283.7 : BOOL; (* S369 M 이송버퍼3 차종6 SP1 *)
    S369_M_이송버퍼3_차종6_썬루프 AT %MW10283.4 : BOOL; (* S369 M 이송버퍼3 차종6 썬루프 *)
    S369_M_이송버퍼3_차종6_일반루프 AT %MW10283.3 : BOOL; (* S369 M 이송버퍼3 차종6 일반루프 *)
    S369_M_이송버퍼3_차종6_파노라마루프 AT %MW10283.5 : BOOL; (* S369 M 이송버퍼3 차종6 파노라마루프 *)
    S369_M_이송버퍼3_차종7_DSL AT %MW10283.9 : BOOL; (* S369 M 이송버퍼3 차종7 DSL *)
    S369_M_이송버퍼3_차종7_GSL AT %MW10283.8 : BOOL; (* S369 M 이송버퍼3 차종7 GSL *)
    S369_M_이송버퍼3_차종7_SP1 AT %MW10283.10 : BOOL; (* S369 M 이송버퍼3 차종7 SP1 *)
    S369_M_이송버퍼3_차종7_SP2 AT %MW10283.11 : BOOL; (* S369 M 이송버퍼3 차종7 SP2 *)
    S369_M_이송버퍼3_차종7_SP3 AT %MW10283.12 : BOOL; (* S369 M 이송버퍼3 차종7 SP3 *)
    S369_M_이송버퍼3_차종7_SP4 AT %MW10283.13 : BOOL; (* S369 M 이송버퍼3 차종7 SP4 *)
    S369_M_이송버퍼3_차종7_SP5 AT %MW10283.14 : BOOL; (* S369 M 이송버퍼3 차종7 SP5 *)
    S369_M_이송버퍼3_차종7_SP6 AT %MW10283.15 : BOOL; (* S369 M 이송버퍼3 차종7 SP6 *)
    S369_M_이송버퍼3_차종8_2WD AT %MW10284.0 : BOOL; (* S369 M 이송버퍼3 차종8 2WD *)
    S369_M_이송버퍼3_차종8_4WD AT %MW10284.1 : BOOL; (* S369 M 이송버퍼3 차종8 4WD *)
    S369_M_이송버퍼3_차종8_SP1 AT %MW10284.2 : BOOL; (* S369 M 이송버퍼3 차종8 SP1 *)
    S369_M_이송버퍼3_차종9_MPI AT %MW10284.3 : BOOL; (* S369 M 이송버퍼3 차종9 MPI *)
    S369_M_이송버퍼3_차종9_SP1 AT %MW10284.5 : BOOL; (* S369 M 이송버퍼3 차종9 SP1 *)
    S369_M_이송버퍼3_차종9_SP10 AT %MW10284.14 : BOOL; (* S369 M 이송버퍼3 차종9 SP10 *)
    S369_M_이송버퍼3_차종9_SP11 AT %MW10284.15 : BOOL; (* S369 M 이송버퍼3 차종9 SP11 *)
    S369_M_이송버퍼3_차종9_SP2 AT %MW10284.6 : BOOL; (* S369 M 이송버퍼3 차종9 SP2 *)
    S369_M_이송버퍼3_차종9_SP3 AT %MW10284.7 : BOOL; (* S369 M 이송버퍼3 차종9 SP3 *)
    S369_M_이송버퍼3_차종9_SP4 AT %MW10284.8 : BOOL; (* S369 M 이송버퍼3 차종9 SP4 *)
    S369_M_이송버퍼3_차종9_SP5 AT %MW10284.9 : BOOL; (* S369 M 이송버퍼3 차종9 SP5 *)
    S369_M_이송버퍼3_차종9_SP6 AT %MW10284.10 : BOOL; (* S369 M 이송버퍼3 차종9 SP6 *)
    S369_M_이송버퍼3_차종9_SP7 AT %MW10284.11 : BOOL; (* S369 M 이송버퍼3 차종9 SP7 *)
    S369_M_이송버퍼3_차종9_SP8 AT %MW10284.12 : BOOL; (* S369 M 이송버퍼3 차종9 SP8 *)
    S369_M_이송버퍼3_차종9_SP9 AT %MW10284.13 : BOOL; (* S369 M 이송버퍼3 차종9 SP9 *)
    S369_M_이송버퍼3_차종9_T_GDI AT %MW10284.4 : BOOL; (* S369 M 이송버퍼3 차종9 T GDI *)
    S369_M_이송버퍼3_차종_AS AT %MW10290.9 : BOOL; (* S369 M 이송버퍼3 차종 AS *)
    S369_M_이송버퍼3_차종_OPT1_R_RACK_무 AT %MW10285.3 : BOOL; (* S369 M 이송버퍼3 차종 OPT1 R RACK 무 *)
    S369_M_이송버퍼3_차종_OPT1_R_RACK_유 AT %MW10285.2 : BOOL; (* S369 M 이송버퍼3 차종 OPT1 R RACK 유 *)
    S369_M_이송버퍼3_차종_OPT1_SP1 AT %MW10285.10 : BOOL; (* S369 M 이송버퍼3 차종 OPT1 SP1 *)
    S369_M_이송버퍼3_차종_OPT1_SP2 AT %MW10285.11 : BOOL; (* S369 M 이송버퍼3 차종 OPT1 SP2 *)
    S369_M_이송버퍼3_차종_OPT1_SP3 AT %MW10285.12 : BOOL; (* S369 M 이송버퍼3 차종 OPT1 SP3 *)
    S369_M_이송버퍼3_차종_OPT1_SP4 AT %MW10285.13 : BOOL; (* S369 M 이송버퍼3 차종 OPT1 SP4 *)
    S369_M_이송버퍼3_차종_OPT1_SP5 AT %MW10285.14 : BOOL; (* S369 M 이송버퍼3 차종 OPT1 SP5 *)
    S369_M_이송버퍼3_차종_OPT1_SP6 AT %MW10285.15 : BOOL; (* S369 M 이송버퍼3 차종 OPT1 SP6 *)
    S369_M_이송버퍼3_차종_OPT1_S_REP_EATER_무 AT %MW10285.7 : BOOL; (* S369 M 이송버퍼3 차종 OPT1 S REP EATER 무 *)
    S369_M_이송버퍼3_차종_OPT1_S_REP_EATER_유 AT %MW10285.6 : BOOL; (* S369 M 이송버퍼3 차종 OPT1 S REP EATER 유 *)
    S369_M_이송버퍼3_차종_OPT1_VAN_무 AT %MW10285.9 : BOOL; (* S369 M 이송버퍼3 차종 OPT1 VAN 무 *)
    S369_M_이송버퍼3_차종_OPT1_VAN_유 AT %MW10285.8 : BOOL; (* S369 M 이송버퍼3 차종 OPT1 VAN 유 *)
    S369_M_이송버퍼3_차종_OPT1_슬라이딩_무 AT %MW10285.1 : BOOL; (* S369 M 이송버퍼3 차종 OPT1 슬라이딩 무 *)
    S369_M_이송버퍼3_차종_OPT1_슬라이딩_유 AT %MW10285.0 : BOOL; (* S369 M 이송버퍼3 차종 OPT1 슬라이딩 유 *)
    S369_M_이송버퍼3_차종_OPT1_폴딩_무 AT %MW10285.5 : BOOL; (* S369 M 이송버퍼3 차종 OPT1 폴딩 무 *)
    S369_M_이송버퍼3_차종_OPT1_폴딩_유 AT %MW10285.4 : BOOL; (* S369 M 이송버퍼3 차종 OPT1 폴딩 유 *)
    S369_M_이송버퍼3_차종_OPT2_SP_WORD1 AT %MW10286 : WORD; (* S369 M 이송버퍼3 차종 OPT2 SP WORD1 *)
    S369_M_이송버퍼3_차종_OPT3_SP_WORD2 AT %MW10287 : WORD; (* S369 M 이송버퍼3 차종 OPT3 SP WORD2 *)
    S369_M_이송버퍼3_차종_OPT4_SP_WORD3 AT %MW10288 : WORD; (* S369 M 이송버퍼3 차종 OPT4 SP WORD3 *)
    S369_M_이송버퍼3_차종_OPT5_SP_WORD4 AT %MW10289 : WORD; (* S369 M 이송버퍼3 차종 OPT5 SP WORD4 *)
    S369_M_이송버퍼3_차종_SP1 AT %MW10290.0 : BOOL; (* S369 M 이송버퍼3 차종 SP1 *)
    S369_M_이송버퍼3_차종_SP2 AT %MW10290.1 : BOOL; (* S369 M 이송버퍼3 차종 SP2 *)
    S369_M_이송버퍼3_차종_SP3 AT %MW10290.2 : BOOL; (* S369 M 이송버퍼3 차종 SP3 *)
    S369_M_이송버퍼3_차종_SP4 AT %MW10290.3 : BOOL; (* S369 M 이송버퍼3 차종 SP4 *)
    S369_M_이송버퍼3_차종_SP5 AT %MW10290.4 : BOOL; (* S369 M 이송버퍼3 차종 SP5 *)
    S369_M_이송버퍼3_차종_SP6 AT %MW10290.5 : BOOL; (* S369 M 이송버퍼3 차종 SP6 *)
    S369_M_이송버퍼3_차종_SP7 AT %MW10290.6 : BOOL; (* S369 M 이송버퍼3 차종 SP7 *)
    S369_M_이송버퍼3_차종_SP8 AT %MW10290.7 : BOOL; (* S369 M 이송버퍼3 차종 SP8 *)
    S369_M_이송버퍼3_차종_SP9 AT %MW10290.15 : BOOL; (* S369 M 이송버퍼3 차종 SP9 *)
    S369_M_이송버퍼3_차종_공대차 AT %MW10290.12 : BOOL; (* S369 M 이송버퍼3 차종 공대차 *)
    S369_M_이송버퍼3_차종_공차 AT %MW10290.10 : BOOL; (* S369 M 이송버퍼3 차종 공차 *)
    S369_M_이송버퍼3_차종_무 AT %MW5002.7 : BOOL;
    S369_M_이송버퍼3_차종_불량대차 AT %MW10290.13 : BOOL; (* S369 M 이송버퍼3 차종 불량대차 *)
    S369_M_이송버퍼3_차종_불량차 AT %MW10290.11 : BOOL; (* S369 M 이송버퍼3 차종 불량차 *)
    S369_M_이송버퍼3_차종_비축 AT %MW10290.8 : BOOL; (* S369 M 이송버퍼3 차종 비축 *)
    S369_M_이송버퍼3_차종_유 AT %MW5002.6 : BOOL;
    S369_M_이송버퍼3_차종_취출대차 AT %MW10290.14 : BOOL; (* S369 M 이송버퍼3 차종 취출대차 *)
    S369_M_이송버퍼4_SEQ AT %MW10260 : WORD; (* S369 M 이송버퍼4 SEQ *)
    S369_M_이송버퍼4_VIN_NO_1_2 AT %MW10271 : WORD; (* S369 M 이송버퍼4 VIN NO 1 2 *)
    S369_M_이송버퍼4_VIN_NO_3_4 AT %MW10272 : WORD; (* S369 M 이송버퍼4 VIN NO 3 4 *)
    S369_M_이송버퍼4_VIN_NO_5_6 AT %MW10273 : WORD; (* S369 M 이송버퍼4 VIN NO 5 6 *)
    S369_M_이송버퍼4_VIN_NO_7_8 AT %MW10274 : WORD; (* S369 M 이송버퍼4 VIN NO 7 8 *)
    S369_M_이송버퍼4_VIN_NO_9_10 AT %MW10275 : WORD; (* S369 M 이송버퍼4 VIN NO 9 10 *)
    S369_M_이송버퍼4_도착완료 AT %MW5003.2 : BOOL;
    S369_M_이송버퍼4_제품감지_이상 AT %MW5014.2 : BOOL; (* S369_M_BELT1_제품감지_이상 *)
    S369_M_이송버퍼4_차종1_AX AT %MW10261.0 : BOOL; (* S369 M 이송버퍼4 차종1 AX *)
    S369_M_이송버퍼4_차종1_B AT %MW10261.1 : BOOL; (* S369 M 이송버퍼4 차종1 B *)
    S369_M_이송버퍼4_차종1_C AT %MW10261.2 : BOOL; (* S369 M 이송버퍼4 차종1 C *)
    S369_M_이송버퍼4_차종1_D AT %MW10261.3 : BOOL; (* S369 M 이송버퍼4 차종1 D *)
    S369_M_이송버퍼4_차종1_E AT %MW10261.4 : BOOL; (* S369 M 이송버퍼4 차종1 E *)
    S369_M_이송버퍼4_차종1_F AT %MW10261.5 : BOOL; (* S369 M 이송버퍼4 차종1 F *)
    S369_M_이송버퍼4_차종1_G AT %MW10261.6 : BOOL; (* S369 M 이송버퍼4 차종1 G *)
    S369_M_이송버퍼4_차종1_H AT %MW10261.7 : BOOL; (* S369 M 이송버퍼4 차종1 H *)
    S369_M_이송버퍼4_차종2_3DR AT %MW10261.8 : BOOL; (* S369 M 이송버퍼4 차종2 3DR *)
    S369_M_이송버퍼4_차종2_4DR AT %MW10261.9 : BOOL; (* S369 M 이송버퍼4 차종2 4DR *)
    S369_M_이송버퍼4_차종2_5DR AT %MW10261.10 : BOOL; (* S369 M 이송버퍼4 차종2 5DR *)
    S369_M_이송버퍼4_차종2_SP1 AT %MW10261.12 : BOOL; (* S369 M 이송버퍼4 차종2 SP1 *)
    S369_M_이송버퍼4_차종2_SP2 AT %MW10261.13 : BOOL; (* S369 M 이송버퍼4 차종2 SP2 *)
    S369_M_이송버퍼4_차종2_WGN AT %MW10261.11 : BOOL; (* S369 M 이송버퍼4 차종2 WGN *)
    S369_M_이송버퍼4_차종3_LHD AT %MW10261.14 : BOOL; (* S369 M 이송버퍼4 차종3 LHD *)
    S369_M_이송버퍼4_차종3_RHD AT %MW10261.15 : BOOL; (* S369 M 이송버퍼4 차종3 RHD *)
    S369_M_이송버퍼4_차종4_EEC AT %MW10262.3 : BOOL; (* S369 M 이송버퍼4 차종4 EEC *)
    S369_M_이송버퍼4_차종4_SP1 AT %MW10262.8 : BOOL; (* S369 M 이송버퍼4 차종4 SP1 *)
    S369_M_이송버퍼4_차종4_SP2 AT %MW10262.9 : BOOL; (* S369 M 이송버퍼4 차종4 SP2 *)
    S369_M_이송버퍼4_차종4_SP3 AT %MW10262.11 : BOOL; (* S369 M 이송버퍼4 차종4 SP3 *)
    S369_M_이송버퍼4_차종4_SP4 AT %MW10262.12 : BOOL; (* S369 M 이송버퍼4 차종4 SP4 *)
    S369_M_이송버퍼4_차종4_SP5 AT %MW10262.13 : BOOL; (* S369 M 이송버퍼4 차종4 SP5 *)
    S369_M_이송버퍼4_차종4_SP6 AT %MW10262.14 : BOOL; (* S369 M 이송버퍼4 차종4 SP6 *)
    S369_M_이송버퍼4_차종4_SP7 AT %MW10262.15 : BOOL; (* S369 M 이송버퍼4 차종4 SP7 *)
    S369_M_이송버퍼4_차종4_내수 AT %MW10262.0 : BOOL; (* S369 M 이송버퍼4 차종4 내수 *)
    S369_M_이송버퍼4_차종4_러시아 AT %MW10262.10 : BOOL; (* S369 M 이송버퍼4 차종4 러시아 *)
    S369_M_이송버퍼4_차종4_북미 AT %MW10262.2 : BOOL; (* S369 M 이송버퍼4 차종4 북미 *)
    S369_M_이송버퍼4_차종4_브라질 AT %MW10262.7 : BOOL; (* S369 M 이송버퍼4 차종4 브라질 *)
    S369_M_이송버퍼4_차종4_수출 AT %MW10262.1 : BOOL; (* S369 M 이송버퍼4 차종4 수출 *)
    S369_M_이송버퍼4_차종4_중국 AT %MW10262.6 : BOOL; (* S369 M 이송버퍼4 차종4 중국 *)
    S369_M_이송버퍼4_차종4_중동 AT %MW10262.5 : BOOL; (* S369 M 이송버퍼4 차종4 중동 *)
    S369_M_이송버퍼4_차종4_호주 AT %MW10262.4 : BOOL; (* S369 M 이송버퍼4 차종4 호주 *)
    S369_M_이송버퍼4_차종5_AT AT %MW10263.1 : BOOL; (* S369 M 이송버퍼4 차종5 AT *)
    S369_M_이송버퍼4_차종5_MT AT %MW10263.0 : BOOL; (* S369 M 이송버퍼4 차종5 MT *)
    S369_M_이송버퍼4_차종5_SP1 AT %MW10263.2 : BOOL; (* S369 M 이송버퍼4 차종5 SP1 *)
    S369_M_이송버퍼4_차종6_DSROOF AT %MW10263.6 : BOOL; (* S369 M 이송버퍼4 차종6 DSROOF *)
    S369_M_이송버퍼4_차종6_SP1 AT %MW10263.7 : BOOL; (* S369 M 이송버퍼4 차종6 SP1 *)
    S369_M_이송버퍼4_차종6_썬루프 AT %MW10263.4 : BOOL; (* S369 M 이송버퍼4 차종6 썬루프 *)
    S369_M_이송버퍼4_차종6_일반루프 AT %MW10263.3 : BOOL; (* S369 M 이송버퍼4 차종6 일반루프 *)
    S369_M_이송버퍼4_차종6_파노라마루프 AT %MW10263.5 : BOOL; (* S369 M 이송버퍼4 차종6 파노라마루프 *)
    S369_M_이송버퍼4_차종7_DSL AT %MW10263.9 : BOOL; (* S369 M 이송버퍼4 차종7 DSL *)
    S369_M_이송버퍼4_차종7_GSL AT %MW10263.8 : BOOL; (* S369 M 이송버퍼4 차종7 GSL *)
    S369_M_이송버퍼4_차종7_SP1 AT %MW10263.10 : BOOL; (* S369 M 이송버퍼4 차종7 SP1 *)
    S369_M_이송버퍼4_차종7_SP2 AT %MW10263.11 : BOOL; (* S369 M 이송버퍼4 차종7 SP2 *)
    S369_M_이송버퍼4_차종7_SP3 AT %MW10263.12 : BOOL; (* S369 M 이송버퍼4 차종7 SP3 *)
    S369_M_이송버퍼4_차종7_SP4 AT %MW10263.13 : BOOL; (* S369 M 이송버퍼4 차종7 SP4 *)
    S369_M_이송버퍼4_차종7_SP5 AT %MW10263.14 : BOOL; (* S369 M 이송버퍼4 차종7 SP5 *)
    S369_M_이송버퍼4_차종7_SP6 AT %MW10263.15 : BOOL; (* S369 M 이송버퍼4 차종7 SP6 *)
    S369_M_이송버퍼4_차종8_2WD AT %MW10264.0 : BOOL; (* S369 M 이송버퍼4 차종8 2WD *)
    S369_M_이송버퍼4_차종8_4WD AT %MW10264.1 : BOOL; (* S369 M 이송버퍼4 차종8 4WD *)
    S369_M_이송버퍼4_차종8_SP1 AT %MW10264.2 : BOOL; (* S369 M 이송버퍼4 차종8 SP1 *)
    S369_M_이송버퍼4_차종9_MPI AT %MW10264.3 : BOOL; (* S369 M 이송버퍼4 차종9 MPI *)
    S369_M_이송버퍼4_차종9_SP1 AT %MW10264.5 : BOOL; (* S369 M 이송버퍼4 차종9 SP1 *)
    S369_M_이송버퍼4_차종9_SP10 AT %MW10264.14 : BOOL; (* S369 M 이송버퍼4 차종9 SP10 *)
    S369_M_이송버퍼4_차종9_SP11 AT %MW10264.15 : BOOL; (* S369 M 이송버퍼4 차종9 SP11 *)
    S369_M_이송버퍼4_차종9_SP2 AT %MW10264.6 : BOOL; (* S369 M 이송버퍼4 차종9 SP2 *)
    S369_M_이송버퍼4_차종9_SP3 AT %MW10264.7 : BOOL; (* S369 M 이송버퍼4 차종9 SP3 *)
    S369_M_이송버퍼4_차종9_SP4 AT %MW10264.8 : BOOL; (* S369 M 이송버퍼4 차종9 SP4 *)
    S369_M_이송버퍼4_차종9_SP5 AT %MW10264.9 : BOOL; (* S369 M 이송버퍼4 차종9 SP5 *)
    S369_M_이송버퍼4_차종9_SP6 AT %MW10264.10 : BOOL; (* S369 M 이송버퍼4 차종9 SP6 *)
    S369_M_이송버퍼4_차종9_SP7 AT %MW10264.11 : BOOL; (* S369 M 이송버퍼4 차종9 SP7 *)
    S369_M_이송버퍼4_차종9_SP8 AT %MW10264.12 : BOOL; (* S369 M 이송버퍼4 차종9 SP8 *)
    S369_M_이송버퍼4_차종9_SP9 AT %MW10264.13 : BOOL; (* S369 M 이송버퍼4 차종9 SP9 *)
    S369_M_이송버퍼4_차종9_T_GDI AT %MW10264.4 : BOOL; (* S369 M 이송버퍼4 차종9 T GDI *)
    S369_M_이송버퍼4_차종_AS AT %MW10270.9 : BOOL; (* S369 M 이송버퍼4 차종 AS *)
    S369_M_이송버퍼4_차종_OPT1_R_RACK_무 AT %MW10265.3 : BOOL; (* S369 M 이송버퍼4 차종 OPT1 R RACK 무 *)
    S369_M_이송버퍼4_차종_OPT1_R_RACK_유 AT %MW10265.2 : BOOL; (* S369 M 이송버퍼4 차종 OPT1 R RACK 유 *)
    S369_M_이송버퍼4_차종_OPT1_SP1 AT %MW10265.10 : BOOL; (* S369 M 이송버퍼4 차종 OPT1 SP1 *)
    S369_M_이송버퍼4_차종_OPT1_SP2 AT %MW10265.11 : BOOL; (* S369 M 이송버퍼4 차종 OPT1 SP2 *)
    S369_M_이송버퍼4_차종_OPT1_SP3 AT %MW10265.12 : BOOL; (* S369 M 이송버퍼4 차종 OPT1 SP3 *)
    S369_M_이송버퍼4_차종_OPT1_SP4 AT %MW10265.13 : BOOL; (* S369 M 이송버퍼4 차종 OPT1 SP4 *)
    S369_M_이송버퍼4_차종_OPT1_SP5 AT %MW10265.14 : BOOL; (* S369 M 이송버퍼4 차종 OPT1 SP5 *)
    S369_M_이송버퍼4_차종_OPT1_SP6 AT %MW10265.15 : BOOL; (* S369 M 이송버퍼4 차종 OPT1 SP6 *)
    S369_M_이송버퍼4_차종_OPT1_S_REP_EATER_무 AT %MW10265.7 : BOOL; (* S369 M 이송버퍼4 차종 OPT1 S REP EATER 무 *)
    S369_M_이송버퍼4_차종_OPT1_S_REP_EATER_유 AT %MW10265.6 : BOOL; (* S369 M 이송버퍼4 차종 OPT1 S REP EATER 유 *)
    S369_M_이송버퍼4_차종_OPT1_VAN_무 AT %MW10265.9 : BOOL; (* S369 M 이송버퍼4 차종 OPT1 VAN 무 *)
    S369_M_이송버퍼4_차종_OPT1_VAN_유 AT %MW10265.8 : BOOL; (* S369 M 이송버퍼4 차종 OPT1 VAN 유 *)
    S369_M_이송버퍼4_차종_OPT1_슬라이딩_무 AT %MW10265.1 : BOOL; (* S369 M 이송버퍼4 차종 OPT1 슬라이딩 무 *)
    S369_M_이송버퍼4_차종_OPT1_슬라이딩_유 AT %MW10265.0 : BOOL; (* S369 M 이송버퍼4 차종 OPT1 슬라이딩 유 *)
    S369_M_이송버퍼4_차종_OPT1_폴딩_무 AT %MW10265.5 : BOOL; (* S369 M 이송버퍼4 차종 OPT1 폴딩 무 *)
    S369_M_이송버퍼4_차종_OPT1_폴딩_유 AT %MW10265.4 : BOOL; (* S369 M 이송버퍼4 차종 OPT1 폴딩 유 *)
    S369_M_이송버퍼4_차종_OPT2_SP_WORD1 AT %MW10266 : WORD; (* S369 M 이송버퍼4 차종 OPT2 SP WORD1 *)
    S369_M_이송버퍼4_차종_OPT3_SP_WORD2 AT %MW10267 : WORD; (* S369 M 이송버퍼4 차종 OPT3 SP WORD2 *)
    S369_M_이송버퍼4_차종_OPT4_SP_WORD3 AT %MW10268 : WORD; (* S369 M 이송버퍼4 차종 OPT4 SP WORD3 *)
    S369_M_이송버퍼4_차종_OPT5_SP_WORD4 AT %MW10269 : WORD; (* S369 M 이송버퍼4 차종 OPT5 SP WORD4 *)
    S369_M_이송버퍼4_차종_SP1 AT %MW10270.0 : BOOL; (* S369 M 이송버퍼4 차종 SP1 *)
    S369_M_이송버퍼4_차종_SP2 AT %MW10270.1 : BOOL; (* S369 M 이송버퍼4 차종 SP2 *)
    S369_M_이송버퍼4_차종_SP3 AT %MW10270.2 : BOOL; (* S369 M 이송버퍼4 차종 SP3 *)
    S369_M_이송버퍼4_차종_SP4 AT %MW10270.3 : BOOL; (* S369 M 이송버퍼4 차종 SP4 *)
    S369_M_이송버퍼4_차종_SP5 AT %MW10270.4 : BOOL; (* S369 M 이송버퍼4 차종 SP5 *)
    S369_M_이송버퍼4_차종_SP6 AT %MW10270.5 : BOOL; (* S369 M 이송버퍼4 차종 SP6 *)
    S369_M_이송버퍼4_차종_SP7 AT %MW10270.6 : BOOL; (* S369 M 이송버퍼4 차종 SP7 *)
    S369_M_이송버퍼4_차종_SP8 AT %MW10270.7 : BOOL; (* S369 M 이송버퍼4 차종 SP8 *)
    S369_M_이송버퍼4_차종_SP9 AT %MW10270.15 : BOOL; (* S369 M 이송버퍼4 차종 SP9 *)
    S369_M_이송버퍼4_차종_공대차 AT %MW10270.12 : BOOL; (* S369 M 이송버퍼4 차종 공대차 *)
    S369_M_이송버퍼4_차종_공차 AT %MW10270.10 : BOOL; (* S369 M 이송버퍼4 차종 공차 *)
    S369_M_이송버퍼4_차종_무 AT %MW5002.5 : BOOL;
    S369_M_이송버퍼4_차종_불량대차 AT %MW10270.13 : BOOL; (* S369 M 이송버퍼4 차종 불량대차 *)
    S369_M_이송버퍼4_차종_불량차 AT %MW10270.11 : BOOL; (* S369 M 이송버퍼4 차종 불량차 *)
    S369_M_이송버퍼4_차종_비축 AT %MW10270.8 : BOOL; (* S369 M 이송버퍼4 차종 비축 *)
    S369_M_이송버퍼4_차종_유 AT %MW5002.4 : BOOL;
    S369_M_이송버퍼4_차종_취출대차 AT %MW10270.14 : BOOL; (* S369 M 이송버퍼4 차종 취출대차 *)
    S369_M_자동_START AT %MW5000.5 : BOOL; (* S369 자동운전중 *)
    S369_M_자동_운전중 AT %MW5000.4 : BOOL; (* S369 자동운전중 *)
    S369_M_자동모드 AT %MW5000.1 : BOOL; (* S369 선택 자동모드 *)
    S369_M_전체_컨베어_도착완료 AT %MW5003.0 : BOOL;
    S369_M_총괄_CP_이상 AT %MW5009.7 : BOOL; (* S369 CP OFF 이상 *)
    S369_M_총괄_CT_이상 AT %MW5010.4 : BOOL; (* S369   TACK TIME 이상 *)
    S369_M_총괄_EOCR_이상 AT %MW5009.8 : BOOL; (* S369_M_총괄_EOCR_이상 *)
    S369_M_총괄_INV_이상 AT %MW5009.9 : BOOL; (* S369_M_총괄_INV_이상 *)
    S369_M_총괄_LS_이상 AT %MW5009.15 : BOOL; (* S369 LS 이상 *)
    S369_M_총괄_MATCH_이상 AT %MW5010.0 : BOOL; (* S369 매트SW 이상 *)
    S369_M_총괄_MC_이상 AT %MW5009.13 : BOOL; (* S369_M_총괄_MC_이상 *)
    S369_M_총괄_MOTOR_이상 AT %MW5010.3 : BOOL; (* S369 MOTOR 이상 *)
    S369_M_총괄_NFB_이상 AT %MW5009.11 : BOOL; (* S369 NFB 이상 *)
    S369_M_총괄_ROBOT_이상 AT %MW5010.1 : BOOL; (* S369 ROBOT 이상 *)
    S369_M_총괄_SAFETY_이상 AT %MW5009.2 : BOOL; (* S369_M_총괄_SAFETY_이상 *)
    S369_M_총괄_SRV_이상 AT %MW5009.10 : BOOL; (* S369 SERVO 이상 *)
    S369_M_총괄_공기압_이상 AT %MW5009.3 : BOOL; (* S369 공기압 이상 *)
    S369_M_총괄_비상정지_이상 AT %MW5009.1 : BOOL; (* S369_M_총괄_비상정지_이상 *)
    S369_M_총괄_사양_이상 AT %MW5009.6 : BOOL; (* S369 사양 이상 *)
    S369_M_총괄_오버런_이상 AT %MW5009.12 : BOOL; (* S369 OVER RUN 이상 *)
    S369_M_총괄_용접타점수_이상 AT %MW5010.2 : BOOL; (* S369 용접타점수 이상 *)
    S369_M_총괄_이상 AT %MW5009.0 : BOOL; (* S369_M_총괄_이상 *)
    S369_M_총괄_제품감지_이상 AT %MW5009.4 : BOOL; (* S369 제품감지 이상 *)
    S369_M_총괄_차종_이상 AT %MW5009.5 : BOOL; (* S369 차종 이상 *)
    S369_M_총괄_통신_이상 AT %MW5009.14 : BOOL; (* S369 통신이상 *)
    S369_M_컨베어_MC_이상 AT %MW5023.0 : BOOL;
    S369_M_컨베어_이동가능 AT %MW5107.8 : BOOL;
    S369_M_컨베어_차종무_도착완료 AT %MW5003.1 : BOOL;
    S369_M_콘베어_이동_전진_LS_이상 AT %MW5107.5 : BOOL;
    S369_M_콘베어_이동_전진_보조 AT %MW5107.1 : BOOL;
    S369_M_콘베어_이동_전진단 AT %MW5107.3 : BOOL;
    S369_M_콘베어_이동_조건 AT %MW5107.0 : BOOL;
    S369_M_콘베어_이동_후진_LS_이상 AT %MW5107.6 : BOOL;
    S369_M_콘베어_이동_후진_보조 AT %MW5107.2 : BOOL;
    S369_M_콘베어_이동_후진단 AT %MW5107.4 : BOOL;
    S369_UNLD_M_NODE_6_42_통신_이상 AT %MW5024.1 : BOOL;
    S369_언로딩버퍼_M_BB_MAIN_DATA_전송_MEMO AT %MW9021.8 : BOOL; (* S369_언로딩버퍼 M BB MAIN DATA 전송 MEMO *)
    S369_언로딩버퍼_M_BB_MAIN_DATA_전송_PLS AT %MW9021.9 : BOOL; (* S369_언로딩버퍼 M BB MAIN DATA 전송 PLS *)
    S369_언로딩버퍼_M_BB_MAIN_DATA_전송_SIGN AT %MW9021.10 : BOOL; (* S369_언로딩버퍼 M BB MAIN DATA 전송 SIGN *)
    S369_언로딩버퍼_M_BB_MAIN_DATA_전송_완료 AT %MW9021.11 : BOOL; (* S369_언로딩버퍼 M BB MAIN DATA 전송 완료 *)
    S369_언로딩버퍼_M_DATA_삭제_PLS AT %MW9021.0 : BOOL; (* S369_언로딩버퍼 M DATA 삭제 PLS *)
    S369_언로딩버퍼_M_DATA_삭제_SIGN AT %MW9021.1 : BOOL; (* S369_언로딩버퍼 M DATA 삭제 SIGN *)
    S369_언로딩버퍼_M_DATA_삭제_완료 AT %MW9021.2 : BOOL; (* S369_언로딩버퍼 M DATA 삭제 완료 *)
    S369_전진_ON AT %MW5048.1 : BOOL; (* S369_전진_ON *)
    S369_컨베어_M_DATA_삭제_PLS AT %MW9020.0 : BOOL; (* S369_컨베어 M DATA 삭제 PLS *)
    S369_컨베어_M_DATA_삭제_SIGN AT %MW9020.1 : BOOL; (* S369_컨베어 M DATA 삭제 SIGN *)
    S369_컨베어_M_DATA_삭제_완료 AT %MW9020.2 : BOOL; (* S369_컨베어 M DATA 삭제 완료 *)
    S369_컨베어_M_DATA_전송_MEMO AT %MW9020.8 : BOOL; (* S369_컨베어 M 이송버퍼02 DATA 전송 MEMO *)
    S369_컨베어_M_DATA_전송_PLS AT %MW9020.9 : BOOL; (* S369_컨베어 M 이송버퍼02 DATA 전송 PLS *)
    S369_컨베어_M_DATA_전송_SIGN AT %MW9020.10 : BOOL; (* S369_컨베어 M 이송버퍼02 DATA 전송 SIGN *)
    S369_컨베어_M_DATA_전송_완료 AT %MW9020.11 : BOOL; (* S369_컨베어 M 이송버퍼02 DATA 전송 완료 *)
    S369_후진_ON AT %MW5048.2 : BOOL; (* S369_후진_ON *)
    SRV1_M_CP_OFF_이상 AT %MW356.3 : BOOL; (* 서보반1 CP OFF 이상 *)
    SRV1_M_PS_DC_LOW AT %MW356.2 : BOOL; (* 서보반1 PS저전압 이상 *)
    SRV1_M_SPD_이상 AT %MW356.1 : BOOL; (* 서보반1 SPD 이상 *)
    SRV1_M_총괄_이상 AT %MW356.0 : BOOL; (* SRV1_M_총괄_이상 *)
    SRV1_M_통신_이상 AT %MW356.4 : BOOL; (* SERVO반1 통신이상 *)
    전체_M_CYCLE_정지 AT %MW308.0 : BOOL; (* 전체_M_CYCLE_정지 *)
    전체_M_GATE_비상정지_정상 AT %MW308.4 : BOOL; (* 전체 M GATE 비상정지 정상 *)
    전체_M_GATE_자동기동 AT %MW308.1 : BOOL; (* 전체_M_자동_운전 *)
    전체_M_OPEN_조건 AT %MW308.3 : BOOL; (* 전체_M_OPEN_조건 *)
    전체_M_운전준비_보조 AT %MW308.5 : BOOL;
    전체_M_이상_리셋 AT %MW308.2 : BOOL; (* ALL공정 PB 이상리셋 *)
    전체_OP_M_총괄_비상정지_정상 AT %MW304.2 : BOOL;
    전체_공정_M_총괄_비상정지_정상 AT %MW304.1 : BOOL;
    전체_라인_M_총괄_CP_OFF AT %MW300.7 : BOOL; (* ALL공정 CP OFF 이상총괄 *)
    전체_라인_M_총괄_CT_이상 AT %MW301.4 : BOOL; (* ALL공정 TACK TIME 이상총괄 *)
    전체_라인_M_총괄_EOCR_이상 AT %MW300.8 : BOOL; (* ALL공정 EOCR 이상총괄 *)
    전체_라인_M_총괄_GATE_OPEN_이상 AT %MW301.5 : BOOL; (* ALL공정 GATEBOX 이상총괄 *)
    전체_라인_M_총괄_INV_이상 AT %MW300.9 : BOOL; (* ALL공정 인버터 이상총괄 *)
    전체_라인_M_총괄_LS_이상 AT %MW300.15 : BOOL; (* ALL공정 LS 이상총괄 *)
    전체_라인_M_총괄_MATCH_이상 AT %MW301.0 : BOOL; (* ALL공정 매트SW 이상총괄 *)
    전체_라인_M_총괄_MC_이상 AT %MW300.13 : BOOL; (* ALL공정 MC 이상총괄 *)
    전체_라인_M_총괄_MOTOR_이상 AT %MW301.3 : BOOL; (* ALL공정 MOTOR 이상총괄 *)
    전체_라인_M_총괄_NFB_이상 AT %MW300.11 : BOOL; (* ALL공정 NFB 이상총괄 *)
    전체_라인_M_총괄_PS_DC_LOW AT %MW301.7 : BOOL; (* ALL공정 PS저전압 이상총괄 *)
    전체_라인_M_총괄_ROBOT_이상 AT %MW301.1 : BOOL; (* ALL공정 ROBOT 총괄이상 *)
    전체_라인_M_총괄_SAFETY_이상 AT %MW300.2 : BOOL; (* ALL공정 SAFETY  이상총괄 *)
    전체_라인_M_총괄_SAG_이상 AT %MW301.6 : BOOL; (* ALL공정 SAG 이상총괄 *)
    전체_라인_M_총괄_SPD_이상 AT %MW301.8 : BOOL; (* ALL공정 SPD 이상총괄 *)
    전체_라인_M_총괄_SRV_이상 AT %MW300.10 : BOOL; (* ALL공정 SERVO 이상총괄 *)
    전체_라인_M_총괄_공기압_이상 AT %MW300.3 : BOOL; (* ALL공정 공기압 이상총괄 *)
    전체_라인_M_총괄_비상정지_이상 AT %MW300.1 : BOOL; (* ALL공정 비상정지 이상총괄 *)
    전체_라인_M_총괄_비상정지_정상 AT %MW304.0 : BOOL;
    전체_라인_M_총괄_사양_이상 AT %MW300.6 : BOOL; (* ALL공정 사양 이상총괄 *)
    전체_라인_M_총괄_오버런_이상 AT %MW300.12 : BOOL; (* ALL공정 OVER RUN 이상총괄 *)
    전체_라인_M_총괄_용접타점수_이상 AT %MW301.2 : BOOL; (* ALL공정 용접타점수 이상총괄 *)
    전체_라인_M_총괄_이상 AT %MW300.0 : BOOL; (* ALL공정 총괄이상 *)
    전체_라인_M_총괄_제품감지_이상 AT %MW300.4 : BOOL; (* ALL공정 제품감지 이상총괄 *)
    전체_라인_M_총괄_차종_이상 AT %MW300.5 : BOOL; (* ALL공정 차종 이상총괄 *)
    전체_라인_M_총괄_통신_이상 AT %MW300.14 : BOOL; (* ALL공정 통신 이상총괄 *)
END_VAR
VAR_GLOBAL
    BB_MAIN_I_1차_작업완료 AT %MW83011.5 : BOOL;
    BB_MAIN_I_2차_작업완료 AT %MW83011.6 : BOOL;
    BB_MAIN_I_CYCLE_STOP AT %MW83011.7 : BOOL;
    BB_MAIN_I_SAFETY_이상 AT %MW83010.14 : BOOL;
    BB_MAIN_I_SPARE_진입_OK AT %MW83011.2 : BOOL;
    BB_MAIN_I_불간섭 AT %MW83011.0 : BOOL;
    BB_MAIN_I_비상정지 AT %MW83010.15 : BOOL;
    BB_MAIN_I_수동모드 AT %MW83010.1 : BOOL;
    BB_MAIN_I_운전준비 AT %MW83010.0 : BOOL;
    BB_MAIN_I_이상 AT %MW83010.13 : BOOL;
    BB_MAIN_I_자동기동 AT %MW83010.3 : BOOL;
    BB_MAIN_I_자동모드 AT %MW83010.2 : BOOL;
    BB_MAIN_I_진입_OK AT %MW83011.1 : BOOL;
    BB_MAIN_I_차종_수신완료 AT %MW83011.4 : BOOL;
    BB_MAIN_I_차종_요구 AT %MW83011.3 : BOOL;
    BB_MAIN_I_취출완료 AT %MW83011.9 : BOOL;
    BB_MAIN_I_통신_CHK AT %MW83011.15 : BOOL;
    BB_MAIN_I_행거클램프_완료 AT %MW83011.8 : BOOL;
    BB_MAIN_O_CYCLE_STOP AT %MW93011.7 : BOOL;
    BB_MAIN_O_SAFETY_이상 AT %MW93010.14 : BOOL;
    BB_MAIN_O_SPARE_진입_OK AT %MW93011.2 : BOOL;
    BB_MAIN_O_도착완료 AT %MW93011.6 : BOOL;
    BB_MAIN_O_불간섭 AT %MW93011.0 : BOOL;
    BB_MAIN_O_비상정지 AT %MW93010.15 : BOOL;
    BB_MAIN_O_수동모드 AT %MW93010.1 : BOOL;
    BB_MAIN_O_운전준비 AT %MW93010.0 : BOOL;
    BB_MAIN_O_이상 AT %MW93010.13 : BOOL;
    BB_MAIN_O_자동기동 AT %MW93010.3 : BOOL;
    BB_MAIN_O_자동모드 AT %MW93010.2 : BOOL;
    BB_MAIN_O_작업완료 AT %MW93011.5 : BOOL;
    BB_MAIN_O_진입_OK AT %MW93011.1 : BOOL;
    BB_MAIN_O_차종_수신완료 AT %MW93011.4 : BOOL;
    BB_MAIN_O_차종_요구 AT %MW93011.3 : BOOL;
    BB_MAIN_O_취출가능 AT %MW93011.9 : BOOL;
    BB_MAIN_O_통신_CHK AT %MW93011.15 : BOOL;
    BB_MAIN_O_행거클램프_요구 AT %MW93011.8 : BOOL;
    EGIS_CWS : BOOL;
    EGIS_ON : BOOL; (* 항시ON (임시용) *)
    GB1_7_1_PLC_BOX_CP_TRIP AT %MW87010.15 : BOOL; (* GB1_7_1_PLC_BOX_CP_TRIP *)
    GB1_EPB_비상정지1 AT %MW87012.0 : BOOL; (* GB1_EPB_비상정지1 *)
    GB1_EPB_비상정지2 AT %MW87012.1 : BOOL; (* GB1_EPB_비상정지2 *)
    GB1_PBL_CYCLE_정지 AT %MW87010.1 : BOOL; (* GB1_PBL_CYCLE_정지 *)
    GB1_PBL_CYCLE_정지_LAMP AT %MW97011.1 : BOOL; (* GB1_PBL_CYCLE_정지_LAMP *)
    GB1_PBL_자동_운전 AT %MW87010.0 : BOOL; (* GB1_PBL_자동_운전 *)
    GB1_PBL_자동_운전_LAMP AT %MW97011.0 : BOOL; (* GB1_PBL_자동_운전_LAMP *)
    GB1_PB_이상_리셋 AT %MW87010.2 : BOOL; (* GB1_PB_이상_리셋 *)
    GB1_SAFETY_DOOR_LOCK1 AT %MW87012.8 : BOOL;
    GB1_SAFETY_DOOR_LOOK2 AT %MW87012.9 : BOOL;
    GB1_SAFETY_DOOR_UNLOOK1 AT %MW97013.0 : BOOL; (* GB1_SAFETY_DOOR_UNLOOK1 *)
    GB1_SAFETY_DOOR_UNLOOK2 AT %MW97013.1 : BOOL; (* GB1_SAFETY_DOOR_UNLOOK2 *)
    GB1_TL_GREEN_LAMP AT %MW97011.9 : BOOL; (* GB1_TL_GREEN_LAMP *)
    GB1_TL_RED_LAMP AT %MW97011.8 : BOOL; (* GB1_TL_RED_LAMP *)
    GB2_7_2_PLC_BOX_CP_TRIP AT %MW87020.15 : BOOL; (* GB2_7_2_PLC_BOX_CP_TRIP *)
    GB2_EPB_비상정지1 AT %MW87022.0 : BOOL; (* GB2_EPB_비상정지1 *)
    GB2_EPB_비상정지2 AT %MW87022.1 : BOOL; (* GB2_EPB_비상정지2 *)
    GB2_PBL_CYCLE_정지 AT %MW87020.1 : BOOL; (* GB2_PBL_CYCLE_정지 *)
    GB2_PBL_CYCLE_정지_LAMP AT %MW97021.1 : BOOL; (* GB2_PBL_CYCLE_정지_LAMP *)
    GB2_PBL_자동_운전 AT %MW87020.0 : BOOL; (* GB2_PBL_자동_운전 *)
    GB2_PBL_자동_운전_LAMP AT %MW97021.0 : BOOL; (* GB2_PBL_자동_운전_LAMP *)
    GB2_PB_이상_리셋 AT %MW87020.2 : BOOL; (* GB2_PB_이상_리셋 *)
    GB2_SAFETY_DOOR_LOCK1 AT %MW87022.8 : BOOL; (* GB2_SAFETY_DOOR_LOCK1 *)
    GB2_SAFETY_DOOR_LOOK2 AT %MW87022.9 : BOOL; (* GB2_SAFETY_DOOR_LOOK2 *)
    GB2_SAFETY_DOOR_UNLOOK1 AT %MW97023.0 : BOOL; (* GB2_SAFETY_DOOR_UNLOOK1 *)
    GB2_SAFETY_DOOR_UNLOOK2 AT %MW97023.1 : BOOL; (* GB2_SAFETY_DOOR_UNLOOK2 *)
    GB2_TL_GREEN_LAMP AT %MW97021.9 : BOOL; (* GB2_TL_GREEN_LAMP *)
    GB2_TL_RED_LAMP AT %MW97021.8 : BOOL; (* GB2_TL_RED_LAMP *)
    GB3_7_3_PLC_BOX_CP_TRIP AT %MW87030.15 : BOOL; (* GB3_7_3_PLC_BOX_CP_TRIP *)
    GB3_EPB_비상정지1 AT %MW87032.0 : BOOL; (* GB3_EPB_비상정지1 *)
    GB3_EPB_비상정지2 AT %MW87032.1 : BOOL; (* GB3_EPB_비상정지2 *)
    GB3_PBL_CYCLE_정지 AT %MW87030.1 : BOOL; (* GB3_PBL_CYCLE_정지 *)
    GB3_PBL_CYCLE_정지_LAMP AT %MW97031.1 : BOOL; (* GB3_PBL_CYCLE_정지_LAMP *)
    GB3_PBL_자동_운전 AT %MW87030.0 : BOOL; (* GB3_PBL_자동_운전 *)
    GB3_PBL_자동_운전_LAMP AT %MW97031.0 : BOOL; (* GB3_PBL_자동_운전_LAMP *)
    GB3_PB_이상_리셋 AT %MW87030.2 : BOOL; (* GB3_PB_이상_리셋 *)
    GB3_SAFETY_DOOR_LOCK1 AT %MW87032.8 : BOOL; (* GB3_SAFETY_DOOR_LOCK1 *)
    GB3_SAFETY_DOOR_LOOK2 AT %MW87032.9 : BOOL; (* GB3_SAFETY_DOOR_LOOK2 *)
    GB3_SAFETY_DOOR_UNLOOK1 AT %MW97033.0 : BOOL; (* GB3_SAFETY_DOOR_UNLOOK1 *)
    GB3_SAFETY_DOOR_UNLOOK2 AT %MW97033.1 : BOOL; (* GB3_SAFETY_DOOR_UNLOOK2 *)
    GB3_TL_GREEN_LAMP AT %MW97031.9 : BOOL; (* GB3_TL_GREEN_LAMP *)
    GB3_TL_RED_LAMP AT %MW97031.8 : BOOL; (* GB3_TL_RED_LAMP *)
    GB4_7_11_PLC_BOX_CP_TRIP AT %MW87110.15 : BOOL; (* GB4 7 11 PLC BOX CP TRIP *)
    GB4_7_3_PLC_BOX_CP_TRIP : BOOL; (* GB3_7_3_PLC_BOX_CP_TRIP *)
    GB4_EPB_비상정지1 AT %MW87112.0 : BOOL; (* GB4 EPB 비상정지1 *)
    GB4_EPB_비상정지2 AT %MW87112.1 : BOOL; (* GB4 EPB 비상정지2 *)
    GB4_PBL_CYCLE_정지 AT %MW87110.1 : BOOL; (* GB4 PBL CYCLE 정지 *)
    GB4_PBL_CYCLE_정지_LAMP AT %MW97111.1 : BOOL; (* GB4 PBL CYCLE 정지 LAMP *)
    GB4_PBL_자동_운전 AT %MW87110.0 : BOOL; (* GB4 PBL 자동 운전 *)
    GB4_PBL_자동_운전_LAMP AT %MW97111.0 : BOOL; (* GB4 PBL 자동 운전 LAMP *)
    GB4_PB_이상_리셋 AT %MW87110.2 : BOOL; (* GB4 PB 이상 리셋 *)
    GB4_SAFETY_DOOR_LOCK1 AT %MW87112.8 : BOOL; (* GB4 SAFETY DOOR LOCK1 *)
    GB4_SAFETY_DOOR_LOOK2 AT %MW87112.9 : BOOL; (* GB4 SAFETY DOOR LOCK2 *)
    GB4_SAFETY_DOOR_UNLOOK1 AT %MW97113.0 : BOOL; (* GB4 SAFETY DOOR UNLOOK1 *)
    GB4_SAFETY_DOOR_UNLOOK2 AT %MW97113.1 : BOOL; (* GB4 SAFETY DOOR UNLOOK2 *)
    GB4_TL_GREEN_LAMP AT %MW97111.9 : BOOL; (* GB4 TL GREEN LAMP *)
    GB4_TL_RED_LAMP AT %MW97111.8 : BOOL; (* GB4 TL RED LAMP *)
    GB5_7_11_PLC_BOX_CP_TRIP : BOOL; (* GB4 7 11 PLC BOX CP TRIP *)
    GB5_7_12_PLC_BOX_CP_TRIP AT %MW87120.15 : BOOL; (* GB5 7 12 PLC BOX CP TRIP *)
    GB5_EPB_비상정지1 AT %MW87122.0 : BOOL; (* GB5 EPB 비상정지1 *)
    GB5_EPB_비상정지2 AT %MW87122.1 : BOOL; (* GB5 EPB 비상정지2 *)
    GB5_PBL_CYCLE_정지 AT %MW87120.1 : BOOL; (* GB5 PBL CYCLE 정지 *)
    GB5_PBL_CYCLE_정지_LAMP AT %MW97121.1 : BOOL; (* GB5 PBL CYCLE 정지 LAMP *)
    GB5_PBL_자동_운전 AT %MW87120.0 : BOOL; (* GB5 PBL 자동 운전 *)
    GB5_PBL_자동_운전_LAMP AT %MW97121.0 : BOOL; (* GB5 PBL 자동 운전 LAMP *)
    GB5_PB_이상_리셋 AT %MW87120.2 : BOOL; (* GB5 PB 이상 리셋 *)
    GB5_SAFETY_DOOR_LOCK1 AT %MW87122.8 : BOOL; (* GB5 SAFETY DOOR LOCK1 *)
    GB5_SAFETY_DOOR_LOOK2 AT %MW87122.9 : BOOL; (* GB5 SAFETY DOOR LOCK2 *)
    GB5_SAFETY_DOOR_UNLOOK1 AT %MW97123.0 : BOOL; (* GB5 SAFETY DOOR UNLOOK1 *)
    GB5_SAFETY_DOOR_UNLOOK2 AT %MW97123.1 : BOOL; (* GB5 SAFETY DOOR UNLOOK2 *)
    GB5_TL_GREEN_LAMP AT %MW97121.9 : BOOL; (* GB5 TL GREEN LAMP *)
    GB5_TL_RED_LAMP AT %MW97121.8 : BOOL; (* GB5 TL RED LAMP *)
    HOP_EPB_비상정지1 AT %MW87503.8 : BOOL; (* HOP_EPB_비상정지1 *)
    HOP_EPB_비상정지2 AT %MW87503.9 : BOOL; (* HOP_EPB_비상정지2 *)
    HOP_PBL_362_4_자동_운전_LP AT %MW97502.1 : BOOL; (* HOP_PBL_362_4_자동_운전_LP *)
    HOP_PBL_365_8_자동_운전 AT %MW87500.7 : BOOL; (* HOP_PBL_365_8_자동_운전 *)
    HOP_PBL_365_8_자동_운전_LP AT %MW97502.2 : BOOL; (* HOP_PBL_365_8_자동_운전_LP *)
    HOP_PBL_369_자동_운전 AT %MW87500.10 : BOOL; (* HOP_PBL_369_자동_운전 *)
    HOP_PBL_369_자동_운전_LP AT %MW97502.3 : BOOL; (* HOP_PBL_369_자동_운전_LP *)
    HOP_PBL_운전준비_ON AT %MW87500.0 : BOOL; (* HOP_PBL_운전준비_ON *)
    HOP_PBL_운전준비_ON_LP AT %MW97502.0 : BOOL; (* HOP_PBL_운전준비_ON_LP *)
    HOP_PB_이상_리셋 AT %MW87500.1 : BOOL; (* HOP_PB_이상_리셋 *)
    HOP_PLB_362_4_자동_운전 AT %MW87500.4 : BOOL; (* HOP PLB 362~4 자동기동 *)
    HOP_SPB_램프_테스트 AT %MW87500.11 : BOOL; (* HOP_SPB_램프_테스트 *)
    HOP_SPB_부저_정지 AT %MW87500.12 : BOOL; (* HOP_SPB_부저_정지 *)
    HOP_SSP_362_4_수동_선택 AT %MW87500.3 : BOOL; (* HOP 362~4 수동선택 *)
    HOP_SSP_362_4_자동_선택 AT %MW87500.2 : BOOL; (* HOP 362~4 자동선택 *)
    HOP_SSP_365_8_수동_선택 AT %MW87500.6 : BOOL; (* HOP_SSP_365_8_수동_선택 *)
    HOP_SSP_365_8_자동_선택 AT %MW87500.5 : BOOL; (* HOP_SSP_365_8_자동_선택 *)
    HOP_SSP_369_수동_선택 AT %MW87500.9 : BOOL; (* HOP_SSP_369_수동_선택 *)
    HOP_SSP_369_자동_선택 AT %MW87500.8 : BOOL; (* HOP_SSP_369_자동_선택 *)
    HOP_부저 AT %MW97502.10 : BOOL; (* HOP_부저 *)
    HOP_타워_빨강_LP AT %MW97502.7 : BOOL; (* HOP_타워_빨강_LP *)
    MCP_DISPLAY_CP_TRIP AT %MW87632.5 : BOOL; (* MCP 출력전원 CP TRIP *)
    MCP_EPB_비상정지1 AT %MW87635.0 : BOOL; (* MCP_EPB_비상정지1 *)
    MCP_EPB_비상정지2 AT %MW87635.1 : BOOL; (* MCP_EPB_비상정지2 *)
    MCP_HUB_CP_TRIP AT %MW87632.0 : BOOL; (* MCP PS1전원  CP TRIP *)
    MCP_INPUT_PWR_CP_TRIP AT %MW87632.2 : BOOL; (* MCP HUB전원  CP TRIP *)
    MCP_OUTPUT_PWR_CP1_TRIP AT %MW87632.3 : BOOL; (* MCP 통신모듈 전원 CP TRIP *)
    MCP_OUTPUT_PWR_CP2_TRIP AT %MW87632.4 : BOOL; (* MCP 입력전원 CP TRIP *)
    MCP_PBL_362_4_자동_운전 AT %MW87630.4 : BOOL; (* MCP PBL 362~4 자동기동 *)
    MCP_PBL_362_4_자동_운전_LP AT %MW97633.1 : BOOL; (* MCP PBL 362~4 자동운전중 (램프) *)
    MCP_PBL_365_8_자동_운전 AT %MW87630.7 : BOOL; (* MCP PBL 365~8 자동기동 *)
    MCP_PBL_365_8_자동_운전_LP AT %MW97633.2 : BOOL; (* MCP PBL 365~8 자동운전중 (램프) *)
    MCP_PBL_369_자동_운전 AT %MW87630.10 : BOOL; (* MCP PBL 369~-1 자동기동 *)
    MCP_PBL_369_자동_운전_LP AT %MW97633.3 : BOOL; (* MCP PBL 369~-1 자동운전중 (램프) *)
    MCP_PBL_운전준비_ON AT %MW87630.0 : BOOL; (* MCP_PBL_운전준비_ON *)
    MCP_PBL_운전준비_ON_LP AT %MW97633.0 : BOOL; (* MCP PBL 운전준비ON (램프) *)
    MCP_PB_이상_리셋 AT %MW87630.1 : BOOL; (* MCP PB 이상리셋 *)
    MCP_PS1_DC_OK AT %MW87631.12 : BOOL; (* MCP PS1 전원 정상 *)
    MCP_PS2_DC_OK AT %MW87631.13 : BOOL; (* MCP PS2 전원 정상 *)
    MCP_PS3_DC_OK AT %MW87631.14 : BOOL; (* MCP PS3 전원 정상 *)
    MCP_PS4_DC_OK AT %MW87631.15 : BOOL; (* MCP PS4 전원 정상 *)
    MCP_SAFTY_MC_ON AT %MW87632.9 : BOOL; (* MCP 운전준비 MC 보조접점 *)
    MCP_SPB_램프_테스트 AT %MW87631.2 : BOOL; (* MCP SPB LAMP 테스트 *)
    MCP_SPB_부저_정지 AT %MW87631.3 : BOOL; (* MCP SPB 부저정지 *)
    MCP_SPB_작업완료_RESET AT %MW87631.6 : BOOL; (* MCP_SPB_작업완료_RESET *)
    MCP_SPB_작업완료_SET AT %MW87631.7 : BOOL; (* MCP_SPB_작업완료_SET *)
    MCP_SSP_362_4_수동_선택 AT %MW87630.2 : BOOL; (* MCP 362~4 수동선택 *)
    MCP_SSP_362_4_자동_선택 AT %MW87630.3 : BOOL; (* MCP 362~4 자동동선택 *)
    MCP_SSP_365_8_수동_선택 AT %MW87630.5 : BOOL; (* MCP_SSP_365_8_수동_선택 *)
    MCP_SSP_365_8_자동_선택 AT %MW87630.6 : BOOL; (* MCP_SSP_365_8_자동_선택 *)
    MCP_SSP_369_수동_선택 AT %MW87630.8 : BOOL; (* MCP_SSP_369_수동_선택 *)
    MCP_SSP_369_자동_선택 AT %MW87630.9 : BOOL; (* MCP_SSP_369_자동_선택 *)
    MCP_TL_GREEN_LAMP AT %MW97633.6 : BOOL; (* MCP 타워램프 (녹색) *)
    MCP_스피커_멜로디1 AT %MW97633.8 : BOOL; (* MCP 스피커 멜로디1 (자동기동) *)
    MCP_스피커_멜로디2 AT %MW97633.9 : BOOL; (* MCP 스피커 멜로디2 (주행) *)
    MCP_스피커_멜로디3 AT %MW97633.10 : BOOL; (* MCP 스피커 멜로디3 (이상) *)
    MCP_스피커_멜로디4 AT %MW97633.11 : BOOL; (* MCP 스피커 멜로디4 (경고) *)
    MCP_스피커_멜로디5 AT %MW97633.12 : BOOL; (* MCP 스피커 멜로디5 (SPARE) *)
    MCP_운전준비_MC_ON AT %MW97636.0 : BOOL; (* MCP 운전준비 MC ON *)
    MCP_타워_노랑_LAMP AT %MW97633.5 : BOOL; (* MCP 타워램프 (황색) *)
    MCP_타워_부저 AT %MW97633.7 : BOOL; (* MCP 타워램프 (부저) *)
    MCP_타워_빨강_LAMP AT %MW97633.4 : BOOL; (* MCP 타워램프 (적색) *)
    MCP_통신_CP_TRIP AT %MW87632.1 : BOOL; (* MCP HMI전원  CP TRIP *)
    PWR_SAG1_DSUB1_NOMAL1 AT %MW87631.10 : BOOL; (* MCP SAG장치 정상 *)
    PWR_SAG1_DSUB8_NOMAL2 AT %MW87631.11 : BOOL; (* MCP SAG장치 이상 *)
    PWR_SPD1_NOMAL AT %MW87631.8 : BOOL; (* MCP 동력반 SPD 정상 *)
    R361_1_I_RB_0_5_COMM_CHK AT %MW84013.14 : BOOL; (* R361_1_I_RB_0_5_COMM_CHK *)
    R361_1_I_RB_10차_간섭무 AT %MW84011.9 : BOOL; (* R361_1_I_RB_10차_간섭무 *)
    R361_1_I_RB_11차_간섭무 AT %MW84011.10 : BOOL; (* R361_1_I_RB_11차_간섭무 *)
    R361_1_I_RB_12차_간섭무 AT %MW84011.11 : BOOL; (* R361_1_I_RB_12차_간섭무 *)
    R361_1_I_RB_1차_간섭무 AT %MW84011.0 : BOOL; (* R361_1_I_RB_1차_간섭무 *)
    R361_1_I_RB_1차_작업완료 AT %MW84010.9 : BOOL; (* R361_1_I_RB_1차_작업완료 *)
    R361_1_I_RB_2차_간섭무 AT %MW84011.1 : BOOL; (* R361_1_I_RB_2차_간섭무 *)
    R361_1_I_RB_2차_작업완료 AT %MW84010.10 : BOOL; (* R361_1_I_RB_2차_작업완료 *)
    R361_1_I_RB_3차_간섭무 AT %MW84011.2 : BOOL; (* R361_1_I_RB_3차_간섭무 *)
    R361_1_I_RB_3차_작업완료 AT %MW84010.11 : BOOL; (* R361_1_I_RB_3차_작업완료 *)
    R361_1_I_RB_4차_간섭무 AT %MW84011.3 : BOOL; (* R361_1_I_RB_4차_간섭무 *)
    R361_1_I_RB_4차_작업완료 AT %MW84010.12 : BOOL; (* R361_1_I_RB_4차_작업완료 *)
    R361_1_I_RB_5차_간섭무 AT %MW84011.4 : BOOL; (* R361_1_I_RB_5차_간섭무 *)
    R361_1_I_RB_5차_작업완료 AT %MW84010.13 : BOOL; (* R361_1_I_RB_5차_작업완료 *)
    R361_1_I_RB_6차_간섭무 AT %MW84011.5 : BOOL; (* R361_1_I_RB_6차_간섭무 *)
    R361_1_I_RB_6차_작업완료 AT %MW84010.14 : BOOL; (* R361_1_I_RB_6차_작업완료 *)
    R361_1_I_RB_7차_간섭무 AT %MW84011.6 : BOOL; (* R361_1_I_RB_7차_간섭무 *)
    R361_1_I_RB_7차_작업완료 AT %MW84010.15 : BOOL; (* R361_1_I_RB_7차_작업완료 *)
    R361_1_I_RB_8차_간섭무 AT %MW84011.7 : BOOL; (* R361_1_I_RB_8차_간섭무 *)
    R361_1_I_RB_9차_간섭무 AT %MW84011.8 : BOOL; (* R361_1_I_RB_9차_간섭무 *)
    R361_1_I_RB_AB_NORMAL_선택 AT %MW84010.6 : BOOL; (* R361_1_I_RB_AB_NORMAL_선택 *)
    R361_1_I_RB_GUN1_FIXED_TIP AT %MW84017 : WORD; (* R361_1_I_RB_GUN1_FIXED_TIP *)
    R361_1_I_RB_GUN1_MOVING_TIP AT %MW84016 : WORD; (* R361_1_I_RB_GUN1_MOVING_TIP *)
    R361_1_I_RB_GUN2_FIXED_TIP AT %MW84019 : WORD; (* R361_1_I_RB_GUN2_FIXED_TIP *)
    R361_1_I_RB_GUN2_MOVING_TIP AT %MW84018 : WORD; (* R361_1_I_RB_GUN2_MOVING_TIP *)
    R361_1_I_RB_INPUT AT %MW84010 : ARRAY[0..3] OF WORD; (* R361_1_I_RB_INPUT *)
    R361_1_I_RB_LS_이상 AT %MW84012.11 : BOOL; (* R361_1_I_RB_LS_이상 *)
    R361_1_I_RB_MOTOR_MC_ON AT %MW84013.15 : BOOL; (* R361_1_I_RB_MOTOR_MC_ON *)
    R361_1_I_RB_PLT_UNLOAD_완료 AT %MW84013.11 : BOOL; (* R361_1_I_RB_PLT_UNLOAD_완료 *)
    R361_1_I_RB_PLT_최종UNLOAD_완료 AT %MW84013.12 : BOOL; (* R361_1_I_RB_PLT_최종UNLOAD_완료 *)
    R361_1_I_RB_PROG_ECHO_1 AT %MW84012.0 : BOOL; (* R361_1_I_RB_PROG_ECHO_1 *)
    R361_1_I_RB_PROG_ECHO_128 AT %MW84012.7 : BOOL; (* R361_1_I_RB_PROG_ECHO_128 *)
    R361_1_I_RB_PROG_ECHO_16 AT %MW84012.4 : BOOL; (* R361_1_I_RB_PROG_ECHO_16 *)
    R361_1_I_RB_PROG_ECHO_2 AT %MW84012.1 : BOOL; (* R361_1_I_RB_PROG_ECHO_2 *)
    R361_1_I_RB_PROG_ECHO_32 AT %MW84012.5 : BOOL; (* R361_1_I_RB_PROG_ECHO_32 *)
    R361_1_I_RB_PROG_ECHO_4 AT %MW84012.2 : BOOL; (* R361_1_I_RB_PROG_ECHO_4 *)
    R361_1_I_RB_PROG_ECHO_64 AT %MW84012.6 : BOOL; (* R361_1_I_RB_PROG_ECHO_64 *)
    R361_1_I_RB_PROG_ECHO_8 AT %MW84012.3 : BOOL; (* R361_1_I_RB_PROG_ECHO_8 *)
    R361_1_I_RB_SP3_8 AT %MW84013.8 : BOOL; (* R361_1_I_RB_SP3_8 *)
    R361_1_I_RB_SP3_9 AT %MW84013.9 : BOOL; (* R361_1_I_RB_SP3_9 *)
    R361_1_I_RB_SPARE_WORD_4 AT %MW84014 : WORD; (* R361_1_I_RB_SPARE_WORD_4 *)
    R361_1_I_RB_SP_1_12 AT %MW84011.12 : BOOL; (* R361_1_I_RB_SP_1_12 *)
    R361_1_I_RB_SP_1_13 AT %MW84011.13 : BOOL; (* R361_1_I_RB_SP_1_13 *)
    R361_1_I_RB_SP_1_14 AT %MW84011.14 : BOOL; (* R361_1_I_RB_SP_1_14 *)
    R361_1_I_RB_SP_1_15 AT %MW84011.15 : BOOL; (* R361_1_I_RB_SP_1_15 *)
    R361_1_I_RB_TC_이상 AT %MW84012.8 : BOOL; (* R361_1_I_RB_TC_이상 *)
    R361_1_I_RB_TIP_CHANGE AT %MW84013.13 : BOOL; (* R361_1_I_RB_TIP_CHANGE *)
    R361_1_I_RB_TIP_DRESSING AT %MW84010.7 : BOOL; (* R361_1_I_RB_TIP_DRESSING *)
    R361_1_I_RB__PLT_카운터리셋완료 AT %MW84013.10 : BOOL; (* R361_1_I_RB__PLT_카운터리셋완료 *)
    R361_1_I_RB_공기압_이상 AT %MW84012.9 : BOOL; (* R361_1_I_RB_공기압_이상 *)
    R361_1_I_RB_냉각수_이상 AT %MW84012.10 : BOOL; (* R361_1_I_RB_냉각수_이상 *)
    R361_1_I_RB_비상정지_NC AT %MW84010.8 : BOOL; (* R361_1_I_RB_비상정지_NC *)
    R361_1_I_RB_비전이상 AT %MW84012.14 : BOOL; (* R361_1_I_RB_비전이상 *)
    R361_1_I_RB_상호인터록_INT1 AT %MW84013.0 : BOOL; (* R361_1_I_RB_상호인터록_INT1 *)
    R361_1_I_RB_상호인터록_INT2 AT %MW84013.1 : BOOL; (* R361_1_I_RB_상호인터록_INT2 *)
    R361_1_I_RB_상호인터록_INT3 AT %MW84013.2 : BOOL; (* R361_1_I_RB_상호인터록_INT3 *)
    R361_1_I_RB_상호인터록_INT4 AT %MW84013.3 : BOOL; (* R361_1_I_RB_상호인터록_INT4 *)
    R361_1_I_RB_상호인터록_INT5 AT %MW84013.4 : BOOL; (* R361_1_I_RB_상호인터록_INT5 *)
    R361_1_I_RB_상호인터록_INT6 AT %MW84013.5 : BOOL; (* R361_1_I_RB_상호인터록_INT6 *)
    R361_1_I_RB_상호인터록_INT7 AT %MW84013.6 : BOOL; (* R361_1_I_RB_상호인터록_INT7 *)
    R361_1_I_RB_상호인터록_INT8 AT %MW84013.7 : BOOL; (* R361_1_I_RB_상호인터록_INT8 *)
    R361_1_I_RB_실러이상 AT %MW84012.13 : BOOL; (* R361_1_I_RB_실러이상 *)
    R361_1_I_RB_용접카운터이상 AT %MW84012.15 : BOOL; (* R361_1_I_RB_용접카운터이상 *)
    R361_1_I_RB_용접타점수 AT %MW84015 : WORD; (* R361_1_I_RB_용접타점수 *)
    R361_1_I_RB_운전준비 AT %MW84010.3 : BOOL; (* R361_1_I_RB_운전준비 *)
    R361_1_I_RB_원위치 AT %MW84010.0 : BOOL; (* R361_1_I_RB_원위치 *)
    R361_1_I_RB_이상리셋 AT %MW84010.2 : BOOL; (* R361_1_I_RB_이상리셋 *)
    R361_1_I_RB_자동 AT %MW84010.4 : BOOL; (* R361_1_I_RB_자동 *)
    R361_1_I_RB_자동기동 AT %MW84010.5 : BOOL; (* R361_1_I_RB_자동기동 *)
    R361_1_I_RB_최종_작업완료 AT %MW84010.1 : BOOL; (* R361_1_I_RB_최종_작업완료 *)
    R361_1_I_RB_통신이상 AT %MW84012.12 : BOOL; (* R361_1_I_RB_통신이상 *)
    R361_1_M_I_RB_1차_작업완료 AT %MW20011.2 : BOOL; (* R361_1_M_I_RB_1차_작업완료 *)
    R361_1_M_I_RB_2차_작업완료 AT %MW20011.3 : BOOL; (* R361_1_M_I_RB_2차_작업완료 *)
    R361_1_M_I_RB_3차_작업완료 AT %MW20011.4 : BOOL; (* R361_1_M_I_RB_3차_작업완료 *)
    R361_1_M_I_RB_4차_작업완료 AT %MW20011.5 : BOOL; (* R361_1_M_I_RB_4차_작업완료 *)
    R361_1_M_I_RB_5차_작업완료 AT %MW20011.6 : BOOL; (* R361_1_M_I_RB_5차_작업완료 *)
    R361_1_M_I_RB_6차_작업완료 AT %MW20011.7 : BOOL; (* R361_1_M_I_RB_6차_작업완료 *)
    R361_1_M_I_RB_7차_작업완료 AT %MW20011.8 : BOOL; (* R361_1_M_I_RB_7차_작업완료 *)
    R361_1_M_I_RB_PAUSE_보조 AT %MW20010.5 : BOOL; (* R361_1_M_I_RB_PAUSE_보조 *)
    R361_1_M_I_RB_PLC_RUN_CHK_이상 AT %MW20010.7 : BOOL; (* R361_1_M_I_RB_PLC_RUN_CHK_이상 *)
    R361_1_M_I_RB_간섭무_1 AT %MW20012.0 : BOOL; (* R361_1_M_I_RB_간섭무_1 *)
    R361_1_M_I_RB_간섭무_10 AT %MW20012.9 : BOOL; (* R361_1_M_I_RB_간섭무_10 *)
    R361_1_M_I_RB_간섭무_11 AT %MW20012.10 : BOOL; (* R361_1_M_I_RB_간섭무_11 *)
    R361_1_M_I_RB_간섭무_12 AT %MW20012.11 : BOOL; (* R361_1_M_I_RB_간섭무_12 *)
    R361_1_M_I_RB_간섭무_2 AT %MW20012.1 : BOOL; (* R361_1_M_I_RB_간섭무_2 *)
    R361_1_M_I_RB_간섭무_3 AT %MW20012.2 : BOOL; (* R361_1_M_I_RB_간섭무_3 *)
    R361_1_M_I_RB_간섭무_4 AT %MW20012.3 : BOOL; (* R361_1_M_I_RB_간섭무_4 *)
    R361_1_M_I_RB_간섭무_5 AT %MW20012.4 : BOOL; (* R361_1_M_I_RB_간섭무_5 *)
    R361_1_M_I_RB_간섭무_6 AT %MW20012.5 : BOOL; (* R361_1_M_I_RB_간섭무_6 *)
    R361_1_M_I_RB_간섭무_7 AT %MW20012.6 : BOOL; (* R361_1_M_I_RB_간섭무_7 *)
    R361_1_M_I_RB_간섭무_8 AT %MW20012.7 : BOOL; (* R361_1_M_I_RB_간섭무_8 *)
    R361_1_M_I_RB_간섭무_9 AT %MW20012.8 : BOOL; (* R361_1_M_I_RB_간섭무_9 *)
    R361_1_M_I_RB_비상정지 AT %MW20010.4 : BOOL; (* R361_1_M_I_RB_비상정지 *)
    R361_1_M_I_RB_운전준비 AT %MW20010.0 : BOOL; (* R361_1_M_I_RB_운전준비 *)
    R361_1_M_I_RB_원위치 AT %MW20010.3 : BOOL; (* R361_1_M_I_RB_원위치 *)
    R361_1_M_I_RB_이상 AT %MW20010.2 : BOOL; (* R361_1_M_I_RB_이상 *)
    R361_1_M_I_RB_자동 AT %MW20010.1 : BOOL; (* R361_1_M_I_RB_자동 *)
    R361_1_M_I_RB_최종작업완료 AT %MW20011.0 : BOOL; (* R361_1_M_I_RB_최종작업완료 *)
    R361_1_M_I_RB_프로그램_이상 AT %MW20010.6 : BOOL; (* R361_1_M_I_RB_프로그램_이상 *)
    R361_1_M_O_RB_1_CYCLE_SET AT %MW21010.3 : BOOL; (* R361_1_M_O_RB_1_CYCLE_SET *)
    R361_1_M_O_RB_1_CYCLE_리셋 AT %MW21010.4 : BOOL; (* R361_1_M_O_RB_1_CYCLE_리셋 *)
    R361_1_M_O_RB_1차_작업완료_리셋 AT %MW21012.0 : BOOL; (* R361_1_M_O_RB_1차_작업완료_리셋 *)
    R361_1_M_O_RB_2차_작업완료_리셋 AT %MW21012.1 : BOOL; (* R361_1_M_O_RB_2차_작업완료_리셋 *)
    R361_1_M_O_RB_2차_진입OK AT %MW21011.8 : BOOL; (* R361_1_M_O_RB_2차_진입OK *)
    R361_1_M_O_RB_3차_작업완료_리셋 AT %MW21012.2 : BOOL; (* R361_1_M_O_RB_3차_작업완료_리셋 *)
    R361_1_M_O_RB_3차_진입OK AT %MW21011.9 : BOOL; (* R361_1_M_O_RB_3차_진입OK *)
    R361_1_M_O_RB_4차_작업완료_리셋 AT %MW21012.3 : BOOL; (* R361_1_M_O_RB_4차_작업완료_리셋 *)
    R361_1_M_O_RB_4차_진입OK AT %MW21011.10 : BOOL; (* R361_1_M_O_RB_4차_진입OK *)
    R361_1_M_O_RB_5차_작업완료_리셋 AT %MW21012.4 : BOOL; (* R361_1_M_O_RB_5차_작업완료_리셋 *)
    R361_1_M_O_RB_5차_진입OK AT %MW21011.11 : BOOL; (* R361_1_M_O_RB_5차_진입OK *)
    R361_1_M_O_RB_6차_작업완료_리셋 AT %MW21012.5 : BOOL; (* R361_1_M_O_RB_6차_작업완료_리셋 *)
    R361_1_M_O_RB_6차_진입OK AT %MW21011.12 : BOOL; (* R361_1_M_O_RB_6차_진입OK *)
    R361_1_M_O_RB_7차_작업완료_리셋 AT %MW21012.6 : BOOL; (* R361_1_M_O_RB_7차_작업완료_리셋 *)
    R361_1_M_O_RB_7차_진입OK AT %MW21011.13 : BOOL; (* R361_1_M_O_RB_7차_진입OK *)
    R361_1_M_O_RB_ATD_OK AT %MW21010.6 : BOOL; (* R361_1_M_O_RB_ATD_OK *)
    R361_1_M_O_RB_PLT_10_진입OK AT %MW21013.10 : BOOL; (* R361_1_M_O_RB_PLT_10_진입OK *)
    R361_1_M_O_RB_PLT_11_진입OK AT %MW21013.11 : BOOL; (* R361_1_M_O_RB_PLT_11_진입OK *)
    R361_1_M_O_RB_PLT_12_진입OK AT %MW21013.12 : BOOL; (* R361_1_M_O_RB_PLT_12_진입OK *)
    R361_1_M_O_RB_PLT_1_진입OK AT %MW21013.1 : BOOL; (* R361_1_M_O_RB_PLT_1_진입OK *)
    R361_1_M_O_RB_PLT_2_진입OK AT %MW21013.2 : BOOL; (* R361_1_M_O_RB_PLT_2_진입OK *)
    R361_1_M_O_RB_PLT_3_진입OK AT %MW21013.3 : BOOL; (* R361_1_M_O_RB_PLT_3_진입OK *)
    R361_1_M_O_RB_PLT_4_진입OK AT %MW21013.4 : BOOL; (* R361_1_M_O_RB_PLT_4_진입OK *)
    R361_1_M_O_RB_PLT_5_진입OK AT %MW21013.5 : BOOL; (* R361_1_M_O_RB_PLT_5_진입OK *)
    R361_1_M_O_RB_PLT_6_진입OK AT %MW21013.6 : BOOL; (* R361_1_M_O_RB_PLT_6_진입OK *)
    R361_1_M_O_RB_PLT_7_진입OK AT %MW21013.7 : BOOL; (* R361_1_M_O_RB_PLT_7_진입OK *)
    R361_1_M_O_RB_PLT_8_진입OK AT %MW21013.8 : BOOL; (* R361_1_M_O_RB_PLT_8_진입OK *)
    R361_1_M_O_RB_PLT_9_진입OK AT %MW21013.9 : BOOL; (* R361_1_M_O_RB_PLT_9_진입OK *)
    R361_1_M_O_RB_PLT_카운터리셋_보조 AT %MW21010.10 : BOOL; (* R361_1_M_O_RB_PLT_카운터리셋_보조 *)
    R361_1_M_O_RB_PROG_NO AT %MW21014 : WORD;
    R361_1_M_O_RB_RESTART_OK AT %MW21010.2 : BOOL; (* R361_1_M_O_RB_RESTART_OK *)
    R361_1_M_O_RB_START_OK AT %MW21010.0 : BOOL; (* R361_1_M_O_RB_START_OK *)
    R361_1_M_O_RB_TEST_MODE_5000회 AT %MW21010.12 : BOOL; (* R361_1_M_O_RB_TEST_MODE_5000회 *)
    R361_1_M_O_RB_TIP_교체_시작 AT %MW21010.7 : BOOL; (* R361_1_M_O_RB_TIP_교체_시작 *)
    R361_1_M_O_RB_TIP_교체_완료 AT %MW21010.8 : BOOL; (* R361_1_M_O_RB_TIP_교체_완료 *)
    R361_1_M_O_RB_VIP_MODE AT %MW21010.11 : BOOL; (* R361_1_M_O_RB_VIP_MODE *)
    R361_1_M_O_RB_냉각수_차단_요청 AT %MW21010.9 : BOOL; (* R361_1_M_O_RB_냉각수_차단_요청 *)
    R361_1_M_O_RB_진입OK_AX차종 AT %MW21011.0 : BOOL; (* R361_1_M_O_RB_진입OK_AX차종 *)
    R361_1_M_O_RB_진입OK_B차종 AT %MW21011.1 : BOOL; (* R361_1_M_O_RB_진입OK_B차종 *)
    R361_1_M_O_RB_진입OK_C차종 AT %MW21011.2 : BOOL; (* R361_1_M_O_RB_진입OK_C차종 *)
    R361_1_M_O_RB_진입OK_D차종 AT %MW21011.3 : BOOL; (* R361_1_M_O_RB_진입OK_D차종 *)
    R361_1_M_O_RB_진입OK_E차종 AT %MW21011.4 : BOOL; (* R361_1_M_O_RB_진입OK_E차종 *)
    R361_1_M_O_RB_진입OK_F차종 AT %MW21011.5 : BOOL; (* R361_1_M_O_RB_진입OK_F차종 *)
    R361_1_M_O_RB_진입OK_G차종 AT %MW21011.6 : BOOL; (* R361_1_M_O_RB_진입OK_G차종 *)
    R361_1_M_O_RB_진입OK_H차종 AT %MW21011.7 : BOOL; (* R361_1_M_O_RB_진입OK_H차종 *)
    R361_1_M_O_RB_최종_작업완료_리셋 AT %MW21010.5 : BOOL; (* R361_1_M_O_RB_최종_작업완료_리셋 *)
    R361_1_M_O_RB_프로그램_OK AT %MW21010.1 : BOOL; (* R361_1_M_O_RB_프로그램_OK *)
    R361_1_O_RB_0_5S_통신_CHK AT %MW94013.14 : BOOL; (* R361_1_O_RB_0_5S_통신_CHK *)
    R361_1_O_RB_2차_진입OK AT %MW94011.8 : BOOL; (* R361_1_O_RB_2차_진입OK *)
    R361_1_O_RB_3차_진입OK AT %MW94011.9 : BOOL; (* R361_1_O_RB_3차_진입OK *)
    R361_1_O_RB_4차_진입OK AT %MW94011.10 : BOOL; (* R361_1_O_RB_4차_진입OK *)
    R361_1_O_RB_5차_진입OK AT %MW94011.11 : BOOL; (* R361_1_O_RB_5차_진입OK *)
    R361_1_O_RB_6차_진입OK AT %MW94011.12 : BOOL; (* R361_1_O_RB_6차_진입OK *)
    R361_1_O_RB_7차_진입OK AT %MW94011.13 : BOOL; (* R361_1_O_RB_7차_진입OK *)
    R361_1_O_RB_AX_1차_진입OK AT %MW94011.0 : BOOL; (* R361_1_O_RB_AX_1차_진입OK *)
    R361_1_O_RB_B_1차_진입OK AT %MW94011.1 : BOOL; (* R361_1_O_RB_B_1차_진입OK *)
    R361_1_O_RB_C_1차_진입OK AT %MW94011.2 : BOOL; (* R361_1_O_RB_C_1차_진입OK *)
    R361_1_O_RB_D_1차_진입OK AT %MW94011.3 : BOOL; (* R361_1_O_RB_D_1차_진입OK *)
    R361_1_O_RB_EACH_작업완료_리셋 AT %MW94010.14 : BOOL; (* R361_1_O_RB_EACH_작업완료_리셋 *)
    R361_1_O_RB_EXT_READY AT %MW94010.11 : BOOL; (* R361_1_O_RB_EXT_READY *)
    R361_1_O_RB_E_1차_진입OK AT %MW94011.4 : BOOL; (* R361_1_O_RB_E_1차_진입OK *)
    R361_1_O_RB_F_1차_진입OK AT %MW94011.5 : BOOL; (* R361_1_O_RB_F_1차_진입OK *)
    R361_1_O_RB_GATE_OPEN_NC AT %MW94013.11 : BOOL; (* R361_1_O_RB_GATE_OPEN_NC *)
    R361_1_O_RB_G_1차_진입OK AT %MW94011.6 : BOOL; (* R361_1_O_RB_G_1차_진입OK *)
    R361_1_O_RB_H_1차_진입OK AT %MW94011.7 : BOOL; (* R361_1_O_RB_H_1차_진입OK *)
    R361_1_O_RB_OUTPUT AT %MW94010 : ARRAY[0..3] OF WORD; (* R361_1_O_RB_OUTPUT *)
    R361_1_O_RB_PAUSE_NC AT %MW94010.13 : BOOL; (* R361_1_O_RB_PAUSE_NC *)
    R361_1_O_RB_PLT10_진입OK AT %MW94012.9 : BOOL; (* R361_1_O_RB_PLT10_진입OK *)
    R361_1_O_RB_PLT11_진입OK AT %MW94012.10 : BOOL; (* R361_1_O_RB_PLT11_진입OK *)
    R361_1_O_RB_PLT12_진입OK AT %MW94012.11 : BOOL; (* R361_1_O_RB_PLT12_진입OK *)
    R361_1_O_RB_PLT1_진입OK AT %MW94012.0 : BOOL; (* R361_1_O_RB_PLT1_진입OK *)
    R361_1_O_RB_PLT2_진입OK AT %MW94012.1 : BOOL; (* R361_1_O_RB_PLT2_진입OK *)
    R361_1_O_RB_PLT3_진입OK AT %MW94012.2 : BOOL; (* R361_1_O_RB_PLT3_진입OK *)
    R361_1_O_RB_PLT4_진입OK AT %MW94012.3 : BOOL; (* R361_1_O_RB_PLT4_진입OK *)
    R361_1_O_RB_PLT5_진입OK AT %MW94012.4 : BOOL; (* R361_1_O_RB_PLT5_진입OK *)
    R361_1_O_RB_PLT6_진입OK AT %MW94012.5 : BOOL; (* R361_1_O_RB_PLT6_진입OK *)
    R361_1_O_RB_PLT7_진입OK AT %MW94012.6 : BOOL; (* R361_1_O_RB_PLT7_진입OK *)
    R361_1_O_RB_PLT8_진입OK AT %MW94012.7 : BOOL; (* R361_1_O_RB_PLT8_진입OK *)
    R361_1_O_RB_PLT9_진입OK AT %MW94012.8 : BOOL; (* R361_1_O_RB_PLT9_진입OK *)
    R361_1_O_RB_PLT_카운터_리셋_요구 AT %MW94013.10 : BOOL; (* R361_1_O_RB_PLT_카운터_리셋_요구 *)
    R361_1_O_RB_PROG_선택1 AT %MW94010.0 : BOOL; (* R361_1_O_RB_PROG_선택1 *)
    R361_1_O_RB_PROG_선택128 AT %MW94010.7 : BOOL; (* R361_1_O_RB_PROG_선택128 *)
    R361_1_O_RB_PROG_선택16 AT %MW94010.4 : BOOL; (* R361_1_O_RB_PROG_선택16 *)
    R361_1_O_RB_PROG_선택2 AT %MW94010.1 : BOOL; (* R361_1_O_RB_PROG_선택2 *)
    R361_1_O_RB_PROG_선택32 AT %MW94010.5 : BOOL; (* R361_1_O_RB_PROG_선택32 *)
    R361_1_O_RB_PROG_선택4 AT %MW94010.2 : BOOL; (* R361_1_O_RB_PROG_선택4 *)
    R361_1_O_RB_PROG_선택64 AT %MW94010.6 : BOOL; (* R361_1_O_RB_PROG_선택64 *)
    R361_1_O_RB_PROG_선택8 AT %MW94010.3 : BOOL; (* R361_1_O_RB_PROG_선택8 *)
    R361_1_O_RB_SP_1_14 AT %MW94011.14 : BOOL; (* R361_1_O_RB_SP_1_14 *)
    R361_1_O_RB_SP_1_15 AT %MW94011.15 : BOOL; (* R361_1_O_RB_SP_1_15 *)
    R361_1_O_RB_SP_2_12 AT %MW94012.12 : BOOL; (* R361_1_O_RB_SP_2_12 *)
    R361_1_O_RB_SP_2_13 AT %MW94012.13 : BOOL; (* R361_1_O_RB_SP_2_13 *)
    R361_1_O_RB_SP_2_14 AT %MW94012.14 : BOOL; (* R361_1_O_RB_SP_2_14 *)
    R361_1_O_RB_SP_5000TH_ON AT %MW94012.15 : BOOL; (* R361_1_O_RB_SP_5000TH_ON *)
    R361_1_O_RB_TIP_CHANGE_END AT %MW94013.9 : BOOL; (* R361_1_O_RB_TIP_CHANGE_END *)
    R361_1_O_RB_TIP_CHANGE_START AT %MW94013.8 : BOOL; (* R361_1_O_RB_TIP_CHANGE_START *)
    R361_1_O_RB_TIP_DRESS_SATRT AT %MW94010.12 : BOOL; (* R361_1_O_RB_TIP_DRESS_SATRT *)
    R361_1_O_RB_VIP_MODE AT %MW94013.15 : BOOL; (* R361_1_O_RB_VIP_MODE *)
    R361_1_O_RB_기동 AT %MW94010.9 : BOOL; (* R361_1_O_RB_기동 *)
    R361_1_O_RB_냉각수차단 AT %MW94010.15 : BOOL; (* R361_1_O_RB_냉각수차단 *)
    R361_1_O_RB_부저정지 AT %MW94013.13 : BOOL; (* R361_1_O_RB_부저정지 *)
    R361_1_O_RB_비상정지_NC AT %MW94013.12 : BOOL; (* R361_1_O_RB_비상정지_NC *)
    R361_1_O_RB_상호인터록_INT1 AT %MW94013.0 : BOOL; (* R361_1_O_RB_상호인터록_INT1 *)
    R361_1_O_RB_상호인터록_INT2 AT %MW94013.1 : BOOL; (* R361_1_O_RB_상호인터록_INT2 *)
    R361_1_O_RB_상호인터록_INT3 AT %MW94013.2 : BOOL; (* R361_1_O_RB_상호인터록_INT3 *)
    R361_1_O_RB_상호인터록_INT4 AT %MW94013.3 : BOOL; (* R361_1_O_RB_상호인터록_INT4 *)
    R361_1_O_RB_상호인터록_INT5 AT %MW94013.4 : BOOL; (* R361_1_O_RB_상호인터록_INT5 *)
    R361_1_O_RB_상호인터록_INT6 AT %MW94013.5 : BOOL; (* R361_1_O_RB_상호인터록_INT6 *)
    R361_1_O_RB_상호인터록_INT7 AT %MW94013.6 : BOOL; (* R361_1_O_RB_상호인터록_INT7 *)
    R361_1_O_RB_상호인터록_INT8 AT %MW94013.7 : BOOL; (* R361_1_O_RB_상호인터록_INT8 *)
    R361_1_O_RB_이상_리셋 AT %MW94010.10 : BOOL; (* R361_1_O_RB_이상_리셋 *)
    R361_1_O_RB_작업완료_리셋 AT %MW94010.8 : BOOL; (* R361_1_O_RB_작업완료_리셋 *)
    R361_2_I_RB_0_5_COMM_CHK AT %MW84023.14 : BOOL; (* R361_2_I_RB_0_5_COMM_CHK *)
    R361_2_I_RB_10차_간섭무 AT %MW84021.9 : BOOL; (* R361_2_I_RB_10차_간섭무 *)
    R361_2_I_RB_11차_간섭무 AT %MW84021.10 : BOOL; (* R361_2_I_RB_11차_간섭무 *)
    R361_2_I_RB_12차_간섭무 AT %MW84021.11 : BOOL; (* R361_2_I_RB_12차_간섭무 *)
    R361_2_I_RB_1차_간섭무 AT %MW84021.0 : BOOL; (* R361_2_I_RB_1차_간섭무 *)
    R361_2_I_RB_1차_작업완료 AT %MW84020.9 : BOOL; (* R361_2_I_RB_1차_작업완료 *)
    R361_2_I_RB_2차_간섭무 AT %MW84021.1 : BOOL; (* R361_2_I_RB_2차_간섭무 *)
    R361_2_I_RB_2차_작업완료 AT %MW84020.10 : BOOL; (* R361_2_I_RB_2차_작업완료 *)
    R361_2_I_RB_3차_간섭무 AT %MW84021.2 : BOOL; (* R361_2_I_RB_3차_간섭무 *)
    R361_2_I_RB_3차_작업완료 AT %MW84020.11 : BOOL; (* R361_2_I_RB_3차_작업완료 *)
    R361_2_I_RB_4차_간섭무 AT %MW84021.3 : BOOL; (* R361_2_I_RB_4차_간섭무 *)
    R361_2_I_RB_4차_작업완료 AT %MW84020.12 : BOOL; (* R361_2_I_RB_4차_작업완료 *)
    R361_2_I_RB_5차_간섭무 AT %MW84021.4 : BOOL; (* R361_2_I_RB_5차_간섭무 *)
    R361_2_I_RB_5차_작업완료 AT %MW84020.13 : BOOL; (* R361_2_I_RB_5차_작업완료 *)
    R361_2_I_RB_6차_간섭무 AT %MW84021.5 : BOOL; (* R361_2_I_RB_6차_간섭무 *)
    R361_2_I_RB_6차_작업완료 AT %MW84020.14 : BOOL; (* R361_2_I_RB_6차_작업완료 *)
    R361_2_I_RB_7차_간섭무 AT %MW84021.6 : BOOL; (* R361_2_I_RB_7차_간섭무 *)
    R361_2_I_RB_7차_작업완료 AT %MW84020.15 : BOOL; (* R361_2_I_RB_7차_작업완료 *)
    R361_2_I_RB_8차_간섭무 AT %MW84021.7 : BOOL; (* R361_2_I_RB_8차_간섭무 *)
    R361_2_I_RB_9차_간섭무 AT %MW84021.8 : BOOL; (* R361_2_I_RB_9차_간섭무 *)
    R361_2_I_RB_AB_NORMAL_선택 AT %MW84020.6 : BOOL; (* R361_2_I_RB_AB_NORMAL_선택 *)
    R361_2_I_RB_GUN1_FIXED_TIP AT %MW84027 : WORD; (* R361_2_I_RB_GUN1_FIXED_TIP *)
    R361_2_I_RB_GUN1_MOVING_TIP AT %MW84026 : WORD; (* R361_2_I_RB_GUN1_MOVING_TIP *)
    R361_2_I_RB_GUN2_FIXED_TIP AT %MW84029 : WORD; (* R361_2_I_RB_GUN2_FIXED_TIP *)
    R361_2_I_RB_GUN2_MOVING_TIP AT %MW84028 : WORD; (* R361_2_I_RB_GUN2_MOVING_TIP *)
    R361_2_I_RB_INPUT AT %MW84020 : ARRAY[0..3] OF WORD; (* R361_2_I_RB_INPUT *)
    R361_2_I_RB_LS_이상 AT %MW84022.11 : BOOL; (* R361_2_I_RB_LS_이상 *)
    R361_2_I_RB_MOTOR_MC_ON AT %MW84023.15 : BOOL; (* R361_2_I_RB_MOTOR_MC_ON *)
    R361_2_I_RB_PLT_UNLOAD_완료 AT %MW84023.11 : BOOL; (* R361_2_I_RB_PLT_UNLOAD_완료 *)
    R361_2_I_RB_PLT_최종UNLOAD_완료 AT %MW84023.12 : BOOL; (* R361_2_I_RB_PLT_최종UNLOAD_완료 *)
    R361_2_I_RB_PROG_ECHO_1 AT %MW84022.0 : BOOL; (* R361_2_I_RB_PROG_ECHO_1 *)
    R361_2_I_RB_PROG_ECHO_128 AT %MW84022.7 : BOOL; (* R361_2_I_RB_PROG_ECHO_128 *)
    R361_2_I_RB_PROG_ECHO_16 AT %MW84022.4 : BOOL; (* R361_2_I_RB_PROG_ECHO_16 *)
    R361_2_I_RB_PROG_ECHO_2 AT %MW84022.1 : BOOL; (* R361_2_I_RB_PROG_ECHO_2 *)
    R361_2_I_RB_PROG_ECHO_32 AT %MW84022.5 : BOOL; (* R361_2_I_RB_PROG_ECHO_32 *)
    R361_2_I_RB_PROG_ECHO_4 AT %MW84022.2 : BOOL; (* R361_2_I_RB_PROG_ECHO_4 *)
    R361_2_I_RB_PROG_ECHO_64 AT %MW84022.6 : BOOL; (* R361_2_I_RB_PROG_ECHO_64 *)
    R361_2_I_RB_PROG_ECHO_8 AT %MW84022.3 : BOOL; (* R361_2_I_RB_PROG_ECHO_8 *)
    R361_2_I_RB_SP3_8 AT %MW84023.8 : BOOL; (* R361_2_I_RB_SP3_8 *)
    R361_2_I_RB_SP3_9 AT %MW84023.9 : BOOL; (* R361_2_I_RB_SP3_9 *)
    R361_2_I_RB_SPARE_WORD_4 AT %MW84024 : WORD; (* R361_2_I_RB_SPARE_WORD_4 *)
    R361_2_I_RB_SP_1_12 AT %MW84021.12 : BOOL; (* R361_2_I_RB_SP_1_12 *)
    R361_2_I_RB_SP_1_13 AT %MW84021.13 : BOOL; (* R361_2_I_RB_SP_1_13 *)
    R361_2_I_RB_SP_1_14 AT %MW84021.14 : BOOL; (* R361_2_I_RB_SP_1_14 *)
    R361_2_I_RB_SP_1_15 AT %MW84021.15 : BOOL; (* R361_2_I_RB_SP_1_15 *)
    R361_2_I_RB_TC_이상 AT %MW84022.8 : BOOL; (* R361_2_I_RB_TC_이상 *)
    R361_2_I_RB_TIP_CHANGE AT %MW84023.13 : BOOL; (* R361_2_I_RB_TIP_CHANGE *)
    R361_2_I_RB_TIP_DRESSING AT %MW84020.7 : BOOL; (* R361_2_I_RB_TIP_DRESSING *)
    R361_2_I_RB__PLT_카운터리셋완료 AT %MW84023.10 : BOOL; (* R361_2_I_RB__PLT_카운터리셋완료 *)
    R361_2_I_RB_공기압_이상 AT %MW84022.9 : BOOL; (* R361_2_I_RB_공기압_이상 *)
    R361_2_I_RB_냉각수_이상 AT %MW84022.10 : BOOL; (* R361_2_I_RB_냉각수_이상 *)
    R361_2_I_RB_비상정지_NC AT %MW84020.8 : BOOL; (* R361_2_I_RB_비상정지_NC *)
    R361_2_I_RB_비전이상 AT %MW84022.14 : BOOL; (* R361_2_I_RB_비전이상 *)
    R361_2_I_RB_상호인터록_INT1 AT %MW84023.0 : BOOL; (* R361_2_I_RB_상호인터록_INT1 *)
    R361_2_I_RB_상호인터록_INT2 AT %MW84023.1 : BOOL; (* R361_2_I_RB_상호인터록_INT2 *)
    R361_2_I_RB_상호인터록_INT3 AT %MW84023.2 : BOOL; (* R361_2_I_RB_상호인터록_INT3 *)
    R361_2_I_RB_상호인터록_INT4 AT %MW84023.3 : BOOL; (* R361_2_I_RB_상호인터록_INT4 *)
    R361_2_I_RB_상호인터록_INT5 AT %MW84023.4 : BOOL; (* R361_2_I_RB_상호인터록_INT5 *)
    R361_2_I_RB_상호인터록_INT6 AT %MW84023.5 : BOOL; (* R361_2_I_RB_상호인터록_INT6 *)
    R361_2_I_RB_상호인터록_INT7 AT %MW84023.6 : BOOL; (* R361_2_I_RB_상호인터록_INT7 *)
    R361_2_I_RB_상호인터록_INT8 AT %MW84023.7 : BOOL; (* R361_2_I_RB_상호인터록_INT8 *)
    R361_2_I_RB_실러이상 AT %MW84022.13 : BOOL; (* R361_2_I_RB_실러이상 *)
    R361_2_I_RB_용접카운터이상 AT %MW84022.15 : BOOL; (* R361_2_I_RB_용접카운터이상 *)
    R361_2_I_RB_용접타점수 AT %MW84025 : WORD; (* R361_2_I_RB_용접타점수 *)
    R361_2_I_RB_운전준비 AT %MW84020.3 : BOOL; (* R361_2_I_RB_운전준비 *)
    R361_2_I_RB_원위치 AT %MW84020.0 : BOOL; (* R361_2_I_RB_원위치 *)
    R361_2_I_RB_이상리셋 AT %MW84020.2 : BOOL; (* R361_2_I_RB_이상리셋 *)
    R361_2_I_RB_자동 AT %MW84020.4 : BOOL; (* R361_2_I_RB_자동 *)
    R361_2_I_RB_자동기동 AT %MW84020.5 : BOOL; (* R361_2_I_RB_자동기동 *)
    R361_2_I_RB_최종_작업완료 AT %MW84020.1 : BOOL; (* R361_2_I_RB_최종_작업완료 *)
    R361_2_I_RB_통신이상 AT %MW84022.12 : BOOL; (* R361_2_I_RB_통신이상 *)
    R361_2_M_I_RB_1차_작업완료 AT %MW20021.2 : BOOL; (* R361_2_M_I_RB_1차_작업완료 *)
    R361_2_M_I_RB_2차_작업완료 AT %MW20021.3 : BOOL; (* R361_2_M_I_RB_2차_작업완료 *)
    R361_2_M_I_RB_3차_작업완료 AT %MW20021.4 : BOOL; (* R361_2_M_I_RB_3차_작업완료 *)
    R361_2_M_I_RB_4차_작업완료 AT %MW20021.5 : BOOL; (* R361_2_M_I_RB_4차_작업완료 *)
    R361_2_M_I_RB_5차_작업완료 AT %MW20021.6 : BOOL; (* R361_2_M_I_RB_5차_작업완료 *)
    R361_2_M_I_RB_6차_작업완료 AT %MW20021.7 : BOOL; (* R361_2_M_I_RB_6차_작업완료 *)
    R361_2_M_I_RB_7차_작업완료 AT %MW20021.8 : BOOL; (* R361_2_M_I_RB_7차_작업완료 *)
    R361_2_M_I_RB_PAUSE_보조 AT %MW20020.5 : BOOL; (* R361_2_M_I_RB_PAUSE_보조 *)
    R361_2_M_I_RB_PLC_RUN_CHK_이상 AT %MW20020.7 : BOOL; (* R361_2_M_I_RB_PLC_RUN_CHK_이상 *)
    R361_2_M_I_RB_간섭무_1 AT %MW20022.0 : BOOL; (* R361_2_M_I_RB_간섭무_1 *)
    R361_2_M_I_RB_간섭무_10 AT %MW20022.9 : BOOL; (* R361_2_M_I_RB_간섭무_10 *)
    R361_2_M_I_RB_간섭무_11 AT %MW20022.10 : BOOL; (* R361_2_M_I_RB_간섭무_11 *)
    R361_2_M_I_RB_간섭무_12 AT %MW20022.11 : BOOL; (* R361_2_M_I_RB_간섭무_12 *)
    R361_2_M_I_RB_간섭무_2 AT %MW20022.1 : BOOL; (* R361_2_M_I_RB_간섭무_2 *)
    R361_2_M_I_RB_간섭무_3 AT %MW20022.2 : BOOL; (* R361_2_M_I_RB_간섭무_3 *)
    R361_2_M_I_RB_간섭무_4 AT %MW20022.3 : BOOL; (* R361_2_M_I_RB_간섭무_4 *)
    R361_2_M_I_RB_간섭무_5 AT %MW20022.4 : BOOL; (* R361_2_M_I_RB_간섭무_5 *)
    R361_2_M_I_RB_간섭무_6 AT %MW20022.5 : BOOL; (* R361_2_M_I_RB_간섭무_6 *)
    R361_2_M_I_RB_간섭무_7 AT %MW20022.6 : BOOL; (* R361_2_M_I_RB_간섭무_7 *)
    R361_2_M_I_RB_간섭무_8 AT %MW20022.7 : BOOL; (* R361_2_M_I_RB_간섭무_8 *)
    R361_2_M_I_RB_간섭무_9 AT %MW20022.8 : BOOL; (* R361_2_M_I_RB_간섭무_9 *)
    R361_2_M_I_RB_비상정지 AT %MW20020.4 : BOOL; (* R361_2_M_I_RB_비상정지 *)
    R361_2_M_I_RB_운전준비 AT %MW20020.0 : BOOL; (* R361_2_M_I_RB_운전준비 *)
    R361_2_M_I_RB_원위치 AT %MW20020.3 : BOOL; (* R361_2_M_I_RB_원위치 *)
    R361_2_M_I_RB_이상 AT %MW20020.2 : BOOL; (* R361_2_M_I_RB_이상 *)
    R361_2_M_I_RB_자동 AT %MW20020.1 : BOOL; (* R361_2_M_I_RB_자동 *)
    R361_2_M_I_RB_최종작업완료 AT %MW20021.0 : BOOL; (* R361_2_M_I_RB_최종작업완료 *)
    R361_2_M_I_RB_프로그램_이상 AT %MW20020.6 : BOOL; (* R361_2_M_I_RB_프로그램_이상 *)
    R361_2_M_O_RB_1_CYCLE_SET AT %MW21020.3 : BOOL; (* R361_2_M_O_RB_1_CYCLE_SET *)
    R361_2_M_O_RB_1_CYCLE_리셋 AT %MW21020.4 : BOOL; (* R361_2_M_O_RB_1_CYCLE_리셋 *)
    R361_2_M_O_RB_1차_작업완료_리셋 AT %MW21022.0 : BOOL; (* R361_2_M_O_RB_1차_작업완료_리셋 *)
    R361_2_M_O_RB_2차_작업완료_리셋 AT %MW21022.1 : BOOL; (* R361_2_M_O_RB_2차_작업완료_리셋 *)
    R361_2_M_O_RB_2차_진입OK AT %MW21021.8 : BOOL; (* R361_2_M_O_RB_2차_진입OK *)
    R361_2_M_O_RB_3차_작업완료_리셋 AT %MW21022.2 : BOOL; (* R361_2_M_O_RB_3차_작업완료_리셋 *)
    R361_2_M_O_RB_3차_진입OK AT %MW21021.9 : BOOL; (* R361_2_M_O_RB_3차_진입OK *)
    R361_2_M_O_RB_4차_작업완료_리셋 AT %MW21022.3 : BOOL; (* R361_2_M_O_RB_4차_작업완료_리셋 *)
    R361_2_M_O_RB_4차_진입OK AT %MW21021.10 : BOOL; (* R361_2_M_O_RB_4차_진입OK *)
    R361_2_M_O_RB_5차_작업완료_리셋 AT %MW21022.4 : BOOL; (* R361_2_M_O_RB_5차_작업완료_리셋 *)
    R361_2_M_O_RB_5차_진입OK AT %MW21021.11 : BOOL; (* R361_2_M_O_RB_5차_진입OK *)
    R361_2_M_O_RB_6차_작업완료_리셋 AT %MW21022.5 : BOOL; (* R361_2_M_O_RB_6차_작업완료_리셋 *)
    R361_2_M_O_RB_6차_진입OK AT %MW21021.12 : BOOL; (* R361_2_M_O_RB_6차_진입OK *)
    R361_2_M_O_RB_7차_작업완료_리셋 AT %MW21022.6 : BOOL; (* R361_2_M_O_RB_7차_작업완료_리셋 *)
    R361_2_M_O_RB_7차_진입OK AT %MW21021.13 : BOOL; (* R361_2_M_O_RB_7차_진입OK *)
    R361_2_M_O_RB_ATD_OK AT %MW21020.6 : BOOL; (* R361_2_M_O_RB_ATD_OK *)
    R361_2_M_O_RB_PLT_10_진입OK AT %MW21023.10 : BOOL; (* R361_2_M_O_RB_PLT_10_진입OK *)
    R361_2_M_O_RB_PLT_11_진입OK AT %MW21023.11 : BOOL; (* R361_2_M_O_RB_PLT_11_진입OK *)
    R361_2_M_O_RB_PLT_12_진입OK AT %MW21023.12 : BOOL; (* R361_2_M_O_RB_PLT_12_진입OK *)
    R361_2_M_O_RB_PLT_1_진입OK AT %MW21023.1 : BOOL; (* R361_2_M_O_RB_PLT_1_진입OK *)
    R361_2_M_O_RB_PLT_2_진입OK AT %MW21023.2 : BOOL; (* R361_2_M_O_RB_PLT_2_진입OK *)
    R361_2_M_O_RB_PLT_3_진입OK AT %MW21023.3 : BOOL; (* R361_2_M_O_RB_PLT_3_진입OK *)
    R361_2_M_O_RB_PLT_4_진입OK AT %MW21023.4 : BOOL; (* R361_2_M_O_RB_PLT_4_진입OK *)
    R361_2_M_O_RB_PLT_5_진입OK AT %MW21023.5 : BOOL; (* R361_2_M_O_RB_PLT_5_진입OK *)
    R361_2_M_O_RB_PLT_6_진입OK AT %MW21023.6 : BOOL; (* R361_2_M_O_RB_PLT_6_진입OK *)
    R361_2_M_O_RB_PLT_7_진입OK AT %MW21023.7 : BOOL; (* R361_2_M_O_RB_PLT_7_진입OK *)
    R361_2_M_O_RB_PLT_8_진입OK AT %MW21023.8 : BOOL; (* R361_2_M_O_RB_PLT_8_진입OK *)
    R361_2_M_O_RB_PLT_9_진입OK AT %MW21023.9 : BOOL; (* R361_2_M_O_RB_PLT_9_진입OK *)
    R361_2_M_O_RB_PLT_카운터리셋_보조 AT %MW21020.10 : BOOL; (* R361_2_M_O_RB_PLT_카운터리셋_보조 *)
    R361_2_M_O_RB_PROG_NO AT %MW21024 : WORD;
    R361_2_M_O_RB_RESTART_OK AT %MW21020.2 : BOOL; (* R361_2_M_O_RB_RESTART_OK *)
    R361_2_M_O_RB_START_OK AT %MW21020.0 : BOOL; (* R361_2_M_O_RB_START_OK *)
    R361_2_M_O_RB_TEST_MODE_5000회 AT %MW21020.12 : BOOL; (* R361_2_M_O_RB_TEST_MODE_5000회 *)
    R361_2_M_O_RB_TIP_교체_시작 AT %MW21020.7 : BOOL; (* R361_2_M_O_RB_TIP_교체_시작 *)
    R361_2_M_O_RB_TIP_교체_완료 AT %MW21020.8 : BOOL; (* R361_2_M_O_RB_TIP_교체_완료 *)
    R361_2_M_O_RB_VIP_MODE AT %MW21020.11 : BOOL; (* R361_2_M_O_RB_VIP_MODE *)
    R361_2_M_O_RB_냉각수_차단_요청 AT %MW21020.9 : BOOL; (* R361_2_M_O_RB_냉각수_차단_요청 *)
    R361_2_M_O_RB_진입OK_AX차종 AT %MW21021.0 : BOOL; (* R361_2_M_O_RB_진입OK_AX차종 *)
    R361_2_M_O_RB_진입OK_B차종 AT %MW21021.1 : BOOL; (* R361_2_M_O_RB_진입OK_B차종 *)
    R361_2_M_O_RB_진입OK_C차종 AT %MW21021.2 : BOOL; (* R361_2_M_O_RB_진입OK_C차종 *)
    R361_2_M_O_RB_진입OK_D차종 AT %MW21021.3 : BOOL; (* R361_2_M_O_RB_진입OK_D차종 *)
    R361_2_M_O_RB_진입OK_E차종 AT %MW21021.4 : BOOL; (* R361_2_M_O_RB_진입OK_E차종 *)
    R361_2_M_O_RB_진입OK_F차종 AT %MW21021.5 : BOOL; (* R361_2_M_O_RB_진입OK_F차종 *)
    R361_2_M_O_RB_진입OK_G차종 AT %MW21021.6 : BOOL; (* R361_2_M_O_RB_진입OK_G차종 *)
    R361_2_M_O_RB_진입OK_H차종 AT %MW21021.7 : BOOL; (* R361_2_M_O_RB_진입OK_H차종 *)
    R361_2_M_O_RB_최종_작업완료_리셋 AT %MW21020.5 : BOOL; (* R361_2_M_O_RB_최종_작업완료_리셋 *)
    R361_2_M_O_RB_프로그램_OK AT %MW21020.1 : BOOL; (* R361_2_M_O_RB_프로그램_OK *)
    R361_2_O_RB_0_5S_통신_CHK AT %MW94023.14 : BOOL; (* R361_2_O_RB_0_5S_통신_CHK *)
    R361_2_O_RB_2차_진입OK AT %MW94021.8 : BOOL; (* R361_2_O_RB_2차_진입OK *)
    R361_2_O_RB_3차_진입OK AT %MW94021.9 : BOOL; (* R361_2_O_RB_3차_진입OK *)
    R361_2_O_RB_4차_진입OK AT %MW94021.10 : BOOL; (* R361_2_O_RB_4차_진입OK *)
    R361_2_O_RB_5차_진입OK AT %MW94021.11 : BOOL; (* R361_2_O_RB_5차_진입OK *)
    R361_2_O_RB_6차_진입OK AT %MW94021.12 : BOOL; (* R361_2_O_RB_6차_진입OK *)
    R361_2_O_RB_7차_진입OK AT %MW94021.13 : BOOL; (* R361_2_O_RB_7차_진입OK *)
    R361_2_O_RB_AX_1차_진입OK AT %MW94021.0 : BOOL; (* R361_2_O_RB_AX_1차_진입OK *)
    R361_2_O_RB_B_1차_진입OK AT %MW94021.1 : BOOL; (* R361_2_O_RB_B_1차_진입OK *)
    R361_2_O_RB_C_1차_진입OK AT %MW94021.2 : BOOL; (* R361_2_O_RB_C_1차_진입OK *)
    R361_2_O_RB_D_1차_진입OK AT %MW94021.3 : BOOL; (* R361_2_O_RB_D_1차_진입OK *)
    R361_2_O_RB_EACH_작업완료_리셋 AT %MW94020.14 : BOOL; (* R361_2_O_RB_EACH_작업완료_리셋 *)
    R361_2_O_RB_EXT_READY AT %MW94020.11 : BOOL; (* R361_2_O_RB_EXT_READY *)
    R361_2_O_RB_E_1차_진입OK AT %MW94021.4 : BOOL; (* R361_2_O_RB_E_1차_진입OK *)
    R361_2_O_RB_F_1차_진입OK AT %MW94021.5 : BOOL; (* R361_2_O_RB_F_1차_진입OK *)
    R361_2_O_RB_GATE_OPEN_NC AT %MW94023.11 : BOOL; (* R361_2_O_RB_GATE_OPEN_NC *)
    R361_2_O_RB_G_1차_진입OK AT %MW94021.6 : BOOL; (* R361_2_O_RB_G_1차_진입OK *)
    R361_2_O_RB_H_1차_진입OK AT %MW94021.7 : BOOL; (* R361_2_O_RB_H_1차_진입OK *)
    R361_2_O_RB_OUTPUT AT %MW94020 : ARRAY[0..3] OF WORD; (* R361_2_O_RB_OUTPUT *)
    R361_2_O_RB_PAUSE_NC AT %MW94020.13 : BOOL; (* R361_2_O_RB_PAUSE_NC *)
    R361_2_O_RB_PLT10_진입OK AT %MW94022.9 : BOOL; (* R361_2_O_RB_PLT10_진입OK *)
    R361_2_O_RB_PLT11_진입OK AT %MW94022.10 : BOOL; (* R361_2_O_RB_PLT11_진입OK *)
    R361_2_O_RB_PLT12_진입OK AT %MW94022.11 : BOOL; (* R361_2_O_RB_PLT12_진입OK *)
    R361_2_O_RB_PLT1_진입OK AT %MW94022.0 : BOOL; (* R361_2_O_RB_PLT1_진입OK *)
    R361_2_O_RB_PLT2_진입OK AT %MW94022.1 : BOOL; (* R361_2_O_RB_PLT2_진입OK *)
    R361_2_O_RB_PLT3_진입OK AT %MW94022.2 : BOOL; (* R361_2_O_RB_PLT3_진입OK *)
    R361_2_O_RB_PLT4_진입OK AT %MW94022.3 : BOOL; (* R361_2_O_RB_PLT4_진입OK *)
    R361_2_O_RB_PLT5_진입OK AT %MW94022.4 : BOOL; (* R361_2_O_RB_PLT5_진입OK *)
    R361_2_O_RB_PLT6_진입OK AT %MW94022.5 : BOOL; (* R361_2_O_RB_PLT6_진입OK *)
    R361_2_O_RB_PLT7_진입OK AT %MW94022.6 : BOOL; (* R361_2_O_RB_PLT7_진입OK *)
    R361_2_O_RB_PLT8_진입OK AT %MW94022.7 : BOOL; (* R361_2_O_RB_PLT8_진입OK *)
    R361_2_O_RB_PLT9_진입OK AT %MW94022.8 : BOOL; (* R361_2_O_RB_PLT9_진입OK *)
    R361_2_O_RB_PLT_카운터_리셋_요구 AT %MW94023.10 : BOOL; (* R361_2_O_RB_PLT_카운터_리셋_요구 *)
    R361_2_O_RB_PROG_선택1 AT %MW94020.0 : BOOL; (* R361_2_O_RB_PROG_선택1 *)
    R361_2_O_RB_PROG_선택128 AT %MW94020.7 : BOOL; (* R361_2_O_RB_PROG_선택128 *)
    R361_2_O_RB_PROG_선택16 AT %MW94020.4 : BOOL; (* R361_2_O_RB_PROG_선택16 *)
    R361_2_O_RB_PROG_선택2 AT %MW94020.1 : BOOL; (* R361_2_O_RB_PROG_선택2 *)
    R361_2_O_RB_PROG_선택32 AT %MW94020.5 : BOOL; (* R361_2_O_RB_PROG_선택32 *)
    R361_2_O_RB_PROG_선택4 AT %MW94020.2 : BOOL; (* R361_2_O_RB_PROG_선택4 *)
    R361_2_O_RB_PROG_선택64 AT %MW94020.6 : BOOL; (* R361_2_O_RB_PROG_선택64 *)
    R361_2_O_RB_PROG_선택8 AT %MW94020.3 : BOOL; (* R361_2_O_RB_PROG_선택8 *)
    R361_2_O_RB_SP_1_14 AT %MW94021.14 : BOOL; (* R361_2_O_RB_SP_1_14 *)
    R361_2_O_RB_SP_1_15 AT %MW94021.15 : BOOL; (* R361_2_O_RB_SP_1_15 *)
    R361_2_O_RB_SP_2_12 AT %MW94022.12 : BOOL; (* R361_2_O_RB_SP_2_12 *)
    R361_2_O_RB_SP_2_13 AT %MW94022.13 : BOOL; (* R361_2_O_RB_SP_2_13 *)
    R361_2_O_RB_SP_2_14 AT %MW94022.14 : BOOL; (* R361_2_O_RB_SP_2_14 *)
    R361_2_O_RB_SP_5000TH_ON AT %MW94022.15 : BOOL; (* R361_2_O_RB_SP_5000TH_ON *)
    R361_2_O_RB_TIP_CHANGE_END AT %MW94023.9 : BOOL; (* R361_2_O_RB_TIP_CHANGE_END *)
    R361_2_O_RB_TIP_CHANGE_START AT %MW94023.8 : BOOL; (* R361_2_O_RB_TIP_CHANGE_START *)
    R361_2_O_RB_TIP_DRESS_SATRT AT %MW94020.12 : BOOL; (* R361_2_O_RB_TIP_DRESS_SATRT *)
    R361_2_O_RB_VIP_MODE AT %MW94023.15 : BOOL; (* R361_2_O_RB_VIP_MODE *)
    R361_2_O_RB_기동 AT %MW94020.9 : BOOL; (* R361_2_O_RB_기동 *)
    R361_2_O_RB_냉각수차단 AT %MW94020.15 : BOOL; (* R361_2_O_RB_냉각수차단 *)
    R361_2_O_RB_부저정지 AT %MW94023.13 : BOOL; (* R361_2_O_RB_부저정지 *)
    R361_2_O_RB_비상정지_NC AT %MW94023.12 : BOOL; (* R361_2_O_RB_비상정지_NC *)
    R361_2_O_RB_상호인터록_INT1 AT %MW94023.0 : BOOL; (* R361_2_O_RB_상호인터록_INT1 *)
    R361_2_O_RB_상호인터록_INT2 AT %MW94023.1 : BOOL; (* R361_2_O_RB_상호인터록_INT2 *)
    R361_2_O_RB_상호인터록_INT3 AT %MW94023.2 : BOOL; (* R361_2_O_RB_상호인터록_INT3 *)
    R361_2_O_RB_상호인터록_INT4 AT %MW94023.3 : BOOL; (* R361_2_O_RB_상호인터록_INT4 *)
    R361_2_O_RB_상호인터록_INT5 AT %MW94023.4 : BOOL; (* R361_2_O_RB_상호인터록_INT5 *)
    R361_2_O_RB_상호인터록_INT6 AT %MW94023.5 : BOOL; (* R361_2_O_RB_상호인터록_INT6 *)
    R361_2_O_RB_상호인터록_INT7 AT %MW94023.6 : BOOL; (* R361_2_O_RB_상호인터록_INT7 *)
    R361_2_O_RB_상호인터록_INT8 AT %MW94023.7 : BOOL; (* R361_2_O_RB_상호인터록_INT8 *)
